Fanuc TP program (LS listing): JOB_VAR_ID_GRIP.LS

/PROG  JOB_VAR_ID_GRIP
/ATTR
OWNER		= MNEDITOR;
COMMENT		= "";
PROG_SIZE	= 104955;
CREATE		= DATE 19-07-31  TIME 17:01:20;
MODIFIED	= DATE 26-07-17  TIME 17:40:38;
FILE_NAME	= JOB_VARI;
VERSION		= 0;
LINE_COUNT = 3549;
MEMORY_SIZE	= 106079;
PROTECT		= READ_WRITE;
TCD:  STACK_SIZE	= 0,
      TASK_PRIORITY	= 50,
      TIME_SLICE	= 0,
      BUSY_LAMP_OFF	= 0,
      ABORT_REQUEST	= 0,
      PAUSE_REQUEST	= 0;
DEFAULT_GROUP	= 1,*,*,*,*;
CONTROL_CODE	= 00000000 00000000;
/APPL

AUTO_SINGULARITY_HEADER;
  ENABLE_SINGULARITY_AVOIDANCE   : TRUE;
/MN
   1:  !R[70] is the item number ;
   2:  !R[71] if using previous data ;
   3:  R[196]=AR[1]    ;
   4:  R[197]=AR[2]    ;
   5:  !------------------------- ;
   6:  !Item Select = 102610459 ;
   7:  SELECT R[70]=459,JMP LBL[459] ;
   8:  !Item Select = 102680512 ;
   9:         =512,JMP LBL[512] ;
  10:  !Item Select = 102730745 ;
  11:         =745,JMP LBL[745] ;
  12:  !Item Select = 102730746 ;
  13:         =746,JMP LBL[746] ;
  14:  !Item Select = 102730747 ;
  15:         =3074,JMP LBL[3074] ;
  16:  !Item Select = 102601361 ;
  17:         =1361,JMP LBL[1361] ;
  18:  !Item Select = 102601363 ;
  19:         =1363,JMP LBL[1363] ;
  20:  !Item Select = 102601364 ;
  21:         =1364,JMP LBL[1364] ;
  22:  !Item Select = 102601365 ;
  23:         =1365,JMP LBL[1365] ;
  24:  !Item Select = 102601366 ;
  25:         =1366,JMP LBL[1366] ;
  26:  !Item Select = 102601367 ;
  27:         =1367,JMP LBL[1367] ;
  28:  !Item Select = 102861623 ;
  29:         =1623,JMP LBL[1623] ;
  30:  !Item Select = 102681826 ;
  31:         =1826,JMP LBL[1826] ;
  32:  !Item Select = 102772047 ;
  33:         =2047,JMP LBL[2047] ;
  34:  !Item Select = 102772052 ;
  35:         =2052,JMP LBL[2052] ;
  36:  !Item Select = 103062126 ;
  37:         =2126,JMP LBL[2126] ;
  38:  !Item Select = 102592407 ;
  39:         =2407,JMP LBL[2407] ;
  40:  !Item Select = 102592408 ;
  41:         =2408,JMP LBL[2408] ;
  42:  !Item Select = 101463245 ;
  43:         =3245,JMP LBL[3245] ;
  44:  !Item Select = 102503284 ;
  45:         =3284,JMP LBL[3284] ;
  46:  !Item Select = 102703721 ;
  47:         =3721,JMP LBL[3721] ;
  48:  !Item Select = 102745613 ;
  49:         =5613,JMP LBL[5613] ;
  50:  !Item Select = 103205791 ;
  51:         =5791,JMP LBL[5791] ;
  52:  !Item Select = 100006970 ;
  53:         =6970,JMP LBL[6970] ;
  54:  !Item Select = 101487064 ;
  55:         =7064,JMP LBL[7064] ;
  56:  !Item Select = 101367132 ;
  57:         =7132,JMP LBL[7132] ;
  58:  !Item Select = 101477920 ;
  59:         =7920,JMP LBL[7920] ;
  60:  !Item Select = 101477937 ;
  61:         =7937,JMP LBL[7937] ;
  62:  !Item Select = 101444857 ;
  63:         =4857,JMP LBL[4857] ;
  64:  !Item Select = 103058815 ;
  65:         =8815,JMP LBL[8815] ;
  66:  !Item Select = 103209297 ;
  67:         =9297,JMP LBL[9297] ;
  68:  !Item Select = 102679394 ;
  69:         =9394,JMP LBL[9394] ;
  70:  !Item Select = 100009654 ;
  71:         =9654,JMP LBL[9654] ;
  72:  !Item Select = 1111199990 ;
  73:         =9990,JMP LBL[9990] ;
  74:  !No conditions are met, jump ;
  75:  !to the very end of the program ;
  76:         ELSE,JMP LBL[9999] ;
  77:   ;
  78:  LBL[459] ;
  79:  !--------------------------- ;
  80:  !Slip ;
  81:  !Item 102610459 , Rev D ;
  82:  !Last Modified: 2023-01-30 ;
  83:  !Modified by: Tsuu ;
  84:  !2.02 IN Height ;
  85:  !3.16 IN ID, 4.760 IN OD ;
  86:  !ID Jaw # 1025 ;
  87:  !--------------------------- ;
  88:  IF (R[70]=459) THEN ;
  89:   ;
  90:  !Define Parameters for INF/OTF ;
  91:  !R[105]=AR[1]=100, 2By3 Sheet ;
  92:  !R[105]=AR[1]=200, 3By4 Sheet ;
  93:  CALL JOB_VAR_SETUP(200) ;
  94:   ;
  95:  !--------------------------- ;
  96:  !Define Parameters for Job ;
  97:  !R[85] "INF_JAW_OFFSET"(Hgt) ;
  98:  R[85]=25    ;
  99:  !R[86] "INF_PICK_OFFSET" 50mm/sec ;
 100:  R[86]=13    ;
 101:  !R[87] "MAIN_LOAD_OFFSET" (PRELOA ;
 102:  R[87]=0    ;
 103:  !R[100] "GRIPPER_ID" 3 values ;
 104:  !If =100, ID Grippers Installed ;
 105:  !If =200, OD Grippers Installed ;
 106:  !If =300, OD 45 Degree Grippers ;
 107:  R[100]=100    ;
 108:  !--------------------------- ;
 109:   ;
 110:  !If using previous setup data ;
 111:  IF (R[71]=459) THEN ;
 112:   ;
 113:  !--------------------------- ;
 114:  !1st: Height of Raw piece ;
 115:  R[190]=53.848    ;
 116:  !2nd: Height of Finish piece ;
 117:  R[191]=51.308    ;
 118:  !3rd: Infeed Height Offset ;
 119:  R[192]=(-55)    ;
 120:  !4th: Outfeed Height Offset ;
 121:  R[193]=(-93)    ;
 122:  !--------------------------- ;
 123:   ;
 124:  CALL CREATE_REG(R[190],R[191],R[192],R[193]) ;
 125:   ;
 126:  ENDIF ;
 127:   ;
 128:  !If new loading or offloading pos ;
 129:  !SET R[104] "IMPORT_LOADPOS" ;
 130:  !SET R[104]=1000, Otherwise NO ;
 131:  R[104]=1000    ;
 132:  IF (R[104]=1000) THEN ;
 133:  !R[260]=43, Preload Pos1 ;
 134:  !R[270]=44, Preload PosFinal ;
 135:  !R[300]=53, Offload PosFinal ;
 136:  !PR[43] Pre-Loading Pos1 ;
 137:  CALL CREATE_PR(43,168.572,(-60.923),352.023,67.102,89.464,65.289) ;
 138:  !PR[44] Final Loading Position ;
 139:  CALL CREATE_PR(44,168.534,(-61.13),363.505,67.212,89.464,65.395) ;
 140:  !PR[53] pre-Unloading Position ;
 141:  CALL CREATE_PR(53,(-125.093),95.886,36.656,173.09,(-88.208),(-174.916)) ;
 142:  !PR[54] Final Unloading Position ;
 143:  CALL CREATE_PR(54,(-124.357),95.73,13.108,173.17,(-88.209),(-174.985)) ;
 144:  !PR[56] assitant Unloading preses ;
 145:  CALL CREATE_PR(56,(-133.84),95.467,273.686,(-177.134),(-88.249),175.184) ;
 146:  !PR[57] assitant Unloading preses ;
 147:  CALL CREATE_PR(57,(-135.964),108.085,344.284,(-177.144),(-88.245),175.194) ;
 148:  !PR[58] assitant Unloading preses ;
 149:  CALL CREATE_PR(58,296.854,360.959,378.47,(-91.75),(-.28),88.063) ;
 150:  ENDIF ;
 151:   ;
 152:  !---------------------------- ;
 153:  !SR[1] = "JOB_VAR_ID_GRIP" ;
 154:  !JOB_VAR_COMMON(R[103])'s value ;
 155:  !---------------------------- ;
 156:  !2By3 SR[1] INF, Max 18(Straight) ;
 157:  !R[103]=100 ;
 158:  !2By3 INF 45 Degree Diagonal Shif ;
 159:  !R[103]=110 ;
 160:  !---------------------------- ;
 161:  !3By4 SR[1] INF, Max 36(Straight) ;
 162:  !R[103]=150 ;
 163:  !3By4 INF 45 Degree Diagonal Shif ;
 164:  !R[103]=160 ;
 165:  !---------------------------- ;
 166:  !R[103] "JOB_PROFILE" Selection ;
 167:  R[103]=150    ;
 168:  CALL JOB_VAR_COMMON(R[103]) ;
 169:   ;
 170:  ENDIF ;
 171:   ;
 172:  JMP LBL[9999] ;
 173:   ;
 174:  !Job 102610459 Logic Ends ;
 175:  !--------------------------- ;
 176:   ;
 177:  LBL[512] ;
 178:  !--------------------------- ;
 179:  !Slip Carrier, Lower ;
 180:  !Item 102680512 , Rev A ;
 181:  !Last Modified: 2026-05-15 ;
 182:  !Modified by: Aaron ;
 183:  !3.74 IN Height ;
 184:  !3.150 IN ID, 4.500 IN OD, 6.0 Lb ;
 185:  !ID Jaw # 1010 ;
 186:  !--------------------------- ;
 187:  IF (R[70]=512) THEN ;
 188:   ;
 189:  !Define Parameters for INF/OTF ;
 190:  !R[105]=AR[1]=100, 2By3 Sheet ;
 191:  !R[105]=AR[1]=200, 3By4 Sheet ;
 192:  CALL JOB_VAR_SETUP(100) ;
 193:   ;
 194:  !--------------------------- ;
 195:  !Define Parameters for Job ;
 196:  R[1]=1    ;
 197:  R[2]=0    ;
 198:  R[4]=0    ;
 199:  R[67]=35    ;
 200:  !R[85] "INF_JAW_OFFSET"(Hgt) ;
 201:  R[85]=78.4    ;
 202:  !R[86] "INF_PICK_OFFSET" 50mm/sec ;
 203:  R[86]=10    ;
 204:  !R[87] "MAIN_LOAD_OFFSET" (PRELOA ;
 205:  R[87]=0    ;
 206:  !R[100] "GRIPPER_ID" 3 values ;
 207:  !If =100, ID Grippers Installed ;
 208:  !If =200, OD Grippers Installed ;
 209:  !If =300, OD 45 Degree Grippers ;
 210:  R[100]=100    ;
 211:  !--------------------------- ;
 212:   ;
 213:  !If using previous setup data ;
 214:  IF (R[71]=512) THEN ;
 215:   ;
 216:  !--------------------------- ;
 217:  !1st: Height of Raw piece ;
 218:  R[190]=101    ;
 219:  !2nd: Height of Finish piece ;
 220:  R[191]=95    ;
 221:  !3rd: Infeed Height Offset ;
 222:  R[192]=(-300)    ;
 223:  !4th: Outfeed Height Offset ;
 224:  R[193]=(-295)    ;
 225:  !--------------------------- ;
 226:   ;
 227:  CALL CREATE_REG(R[190],R[191],R[192],R[193]) ;
 228:   ;
 229:  ENDIF ;
 230:   ;
 231:  !If new loading or offloading pos ;
 232:  !SET R[104] "IMPORT_LOADPOS" ;
 233:  !SET R[104]=1000, Otherwise NO ;
 234:  R[104]=1000    ;
 235:  IF (R[104]=1000) THEN ;
 236:  !R[260]=43, Preload Pos1 ;
 237:  !R[270]=44, Preload PosFinal ;
 238:  !R[300]=53, Offload PosFinal ;
 239:  !PR[43] Pre-Loading Pos1 ;
 240:  CALL CREATE_PR(43,168.016,(-60.327),359.452,97.401,89.434,95.565) ;
 241:  !PR[44] Final Loading Position ;
 242:  CALL CREATE_PR(44,168.082,(-60.943),407.633,97.503,89.436,95.659) ;
 243:  !PR[53] pre-Unloading Position ;
 244:  CALL CREATE_PR(53,(-131.438),93.126,204.569,171.755,(-88.248),(-173.108)) ;
 245:  !PR[54] Final Unloading Position ;
 246:  CALL CREATE_PR(54,(-130.24),93.445,164.559,171.759,(-88.249),(-173.121)) ;
 247:  !PR[56] assitant Unloading preses ;
 248:  CALL CREATE_PR(56,(-133.84),95.467,273.686,(-177.134),(-88.249),175.184) ;
 249:  !PR[57] assitant Unloading preses ;
 250:  CALL CREATE_PR(57,(-135.964),108.085,344.284,(-177.144),(-88.245),175.194) ;
 251:  !PR[58] assitant Unloading preses ;
 252:  CALL CREATE_PR(58,296.854,360.959,378.47,(-91.75),(-.28),88.063) ;
 253:  ENDIF ;
 254:   ;
 255:  !---------------------------- ;
 256:  !SR[1] = "JOB_VAR_ID_GRIP" ;
 257:  !JOB_VAR_COMMON(R[103])'s value ;
 258:  !---------------------------- ;
 259:  !2By3 SR[1] INF, Max 18(Straight) ;
 260:  !R[103]=100 ;
 261:  !2By3 INF 45 Degree Diagonal Shif ;
 262:  !R[103]=110 ;
 263:  !---------------------------- ;
 264:  !3By4 SR[1] INF, Max 36(Straight) ;
 265:  !R[103]=150 ;
 266:  !3By4 INF 45 Degree Diagonal Shif ;
 267:  !R[103]=160 ;
 268:  !---------------------------- ;
 269:  !R[103] "JOB_PROFILE" Selection ;
 270:  R[103]=100    ;
 271:  CALL JOB_VAR_COMMON(R[103]) ;
 272:   ;
 273:  ENDIF ;
 274:   ;
 275:  JMP LBL[9999] ;
 276:   ;
 277:  !Job 102680512 Logic Ends ;
 278:  !--------------------------- ;
 279:   ;
 280:  LBL[745] ;
 281:  !--------------------------- ;
 282:  !Top Slip Support, Packer ;
 283:  !Item 102730745 , Rev A ;
 284:  !Last Modified: 2026-02-04 ;
 285:  !Modified by: Aaron ;
 286:  !4.705 IN Height ;
 287:  !3.4 IN ID, 4.18 IN OD, 18.5 Lbs ;
 288:  !ID Jaw # 1016 ;
 289:  !--------------------------- ;
 290:  IF (R[70]=745) THEN ;
 291:   ;
 292:  !Define Parameters for INF/OTF ;
 293:  !R[105]=AR[1]=100, 2By3 Sheet ;
 294:  !R[105]=AR[1]=200, 3By4 Sheet ;
 295:  CALL JOB_VAR_SETUP(100) ;
 296:   ;
 297:  !--------------------------- ;
 298:  !Define Parameters for Job ;
 299:  R[1]=1    ;
 300:  R[2]=1    ;
 301:  R[4]=0    ;
 302:  R[67]=45    ;
 303:  !R[85] "INF_JAW_OFFSET"(Hgt) ;
 304:  R[85]=20    ;
 305:  !R[86] "INF_PICK_OFFSET" 50mm/sec ;
 306:  R[86]=2    ;
 307:  !R[87] "MAIN_LOAD_OFFSET" (PRELOA ;
 308:  R[87]=0    ;
 309:  !R[100] "GRIPPER_ID" 3 values ;
 310:  !If =100, ID Grippers Installed ;
 311:  !If =200, OD Grippers Installed ;
 312:  !If =300, OD 45 Degree Grippers ;
 313:  R[100]=100    ;
 314:  !--------------------------- ;
 315:   ;
 316:  !If using previous setup data ;
 317:  IF (R[71]=745) THEN ;
 318:   ;
 319:  !--------------------------- ;
 320:  !1st: Height of Raw piece ;
 321:  R[190]=124.8    ;
 322:  !2nd: Height of Finish piece ;
 323:  R[191]=119.51    ;
 324:  !3rd: Infeed Height Offset ;
 325:  R[192]=(-298)    ;
 326:  !4th: Outfeed Height Offset ;
 327:  R[193]=(-250)    ;
 328:  !--------------------------- ;
 329:   ;
 330:  CALL CREATE_REG(R[190],R[191],R[192],R[193]) ;
 331:   ;
 332:  ENDIF ;
 333:   ;
 334:  !If new loading or offloading pos ;
 335:  !SET R[104] "IMPORT_LOADPOS" ;
 336:  !SET R[104]=1000, Otherwise NO ;
 337:  R[104]=1000    ;
 338:  IF (R[104]=1000) THEN ;
 339:  !R[260]=43, Preload Pos1 ;
 340:  !R[270]=44, Preload PosFinal ;
 341:  !R[300]=53, Offload PosFinal ;
 342:  !PR[43] Pre-Loading Pos1 ;
 343:  CALL CREATE_PR(43,163.322,(-60.984),274.82,151.418,88.347,149.991) ;
 344:  !PR[44] Final Loading Position ;
 345:  CALL CREATE_PR(44,164.891,(-62.061),335.467,151.455,88.338,150.017) ;
 346:  !PR[53] pre-Unloading Position ;
 347:  CALL CREATE_PR(53,(-130.787),93.777,177.177,170.605,(-88.218),(-171.87)) ;
 348:  !PR[54] Final Unloading Position ;
 349:  CALL CREATE_PR(54,(-127.959),94.047,84.786,170.695,(-88.22),(-171.955)) ;
 350:  !PR[56] assitant Unloading preses ;
 351:  CALL CREATE_PR(56,(-133.84),95.467,273.686,(-177.134),(-88.249),175.184) ;
 352:  !PR[57] assitant Unloading preses ;
 353:  CALL CREATE_PR(57,(-135.964),108.085,344.284,(-177.144),(-88.245),175.194) ;
 354:  !PR[58] assitant Unloading preses ;
 355:  CALL CREATE_PR(58,296.854,360.959,378.47,(-91.75),(-.28),88.063) ;
 356:  ENDIF ;
 357:   ;
 358:  !---------------------------- ;
 359:  !SR[1] = "JOB_VAR_ID_GRIP" ;
 360:  !JOB_VAR_COMMON(R[103])'s value ;
 361:  !---------------------------- ;
 362:  !2By3 SR[1] INF, Max 18(Straight) ;
 363:  !R[103]=100 ;
 364:  !2By3 INF 45 Degree Diagonal Shif ;
 365:  !R[103]=110 ;
 366:  !---------------------------- ;
 367:  !3By4 SR[1] INF, Max 36(Straight) ;
 368:  !R[103]=150 ;
 369:  !3By4 INF 45 Degree Diagonal Shif ;
 370:  !R[103]=160 ;
 371:  !---------------------------- ;
 372:  !R[103] "JOB_PROFILE" Selection ;
 373:  R[103]=100    ;
 374:  CALL JOB_VAR_COMMON(R[103]) ;
 375:   ;
 376:  ENDIF ;
 377:   ;
 378:  JMP LBL[9999] ;
 379:   ;
 380:  !Job 102730745 Logic Ends ;
 381:  !--------------------------- ;
 382:   ;
 383:  LBL[746] ;
 384:  !--------------------------- ;
 385:  !Wedge, Top ;
 386:  !Item 102730746 , Rev A ;
 387:  !Last Modified: 2026-05-04 ;
 388:  !Modified by: Aaron ;
 389:  !1.88 IN Height ;
 390:  !3.4 IN ID, 4.32 IN OD, 6.0 Lbs W ;
 391:  !ID Jaw # 1010 ;
 392:  !--------------------------- ;
 393:  IF (R[70]=746) THEN ;
 394:   ;
 395:  !Define Parameters for INF/OTF ;
 396:  !R[105]=AR[1]=100, 2By3 Sheet ;
 397:  !R[105]=AR[1]=200, 3By4 Sheet ;
 398:  CALL JOB_VAR_SETUP(100) ;
 399:   ;
 400:  !--------------------------- ;
 401:  !Define Parameters for Job ;
 402:  R[1]=1    ;
 403:  R[2]=1    ;
 404:  R[4]=0    ;
 405:  R[67]=10    ;
 406:  !R[85] "INF_JAW_OFFSET"(Hgt) ;
 407:  R[85]=94.4    ;
 408:  !R[86] "INF_PICK_OFFSET" 50mm/sec ;
 409:  R[86]=30    ;
 410:  !R[87] "MAIN_LOAD_OFFSET" (PRELOA ;
 411:  R[87]=0    ;
 412:  !R[100] "GRIPPER_ID" 3 values ;
 413:  !If =100, ID Grippers Installed ;
 414:  !If =200, OD Grippers Installed ;
 415:  !If =300, OD 45 Degree Grippers ;
 416:  R[100]=100    ;
 417:  !--------------------------- ;
 418:   ;
 419:  !If using previous setup data ;
 420:  IF (R[71]=746) THEN ;
 421:   ;
 422:  !--------------------------- ;
 423:  !1st: Height of Raw piece ;
 424:  R[190]=53.5    ;
 425:  !2nd: Height of Finish piece ;
 426:  R[191]=47.75    ;
 427:  !3rd: Infeed Height Offset ;
 428:  R[192]=(-300)    ;
 429:  !4th: Outfeed Height Offset ;
 430:  R[193]=(-295)    ;
 431:  !--------------------------- ;
 432:   ;
 433:  CALL CREATE_REG(R[190],R[191],R[192],R[193]) ;
 434:   ;
 435:  ENDIF ;
 436:   ;
 437:  !If new loading or offloading pos ;
 438:  !SET R[104] "IMPORT_LOADPOS" ;
 439:  !SET R[104]=1000, Otherwise NO ;
 440:  R[104]=1000    ;
 441:  IF (R[104]=1000) THEN ;
 442:  !R[260]=43, Preload Pos1 ;
 443:  !R[270]=44, Preload PosFinal ;
 444:  !R[300]=53, Offload PosFinal ;
 445:  !PR[43] Pre-Loading Pos1 ;
 446:  CALL CREATE_PR(43,168.016,(-60.327),359.452,97.401,89.434,95.565) ;
 447:  !PR[44] Final Loading Position ;
 448:  CALL CREATE_PR(44,168.082,(-60.943),407.633,97.503,89.436,95.659) ;
 449:  !PR[53] pre-Unloading Position ;
 450:  CALL CREATE_PR(53,(-131.438),93.126,204.569,171.755,(-88.248),(-173.108)) ;
 451:  !PR[54] Final Unloading Position ;
 452:  CALL CREATE_PR(54,(-130.24),93.445,164.559,171.759,(-88.249),(-173.121)) ;
 453:  !PR[56] assitant Unloading preses ;
 454:  CALL CREATE_PR(56,(-133.84),95.467,273.686,(-177.134),(-88.249),175.184) ;
 455:  !PR[57] assitant Unloading preses ;
 456:  CALL CREATE_PR(57,(-135.964),108.085,344.284,(-177.144),(-88.245),175.194) ;
 457:  !PR[58] assitant Unloading preses ;
 458:  CALL CREATE_PR(58,296.854,360.959,378.47,(-91.75),(-.28),88.063) ;
 459:  ENDIF ;
 460:   ;
 461:  !---------------------------- ;
 462:  !SR[1] = "JOB_VAR_ID_GRIP" ;
 463:  !JOB_VAR_COMMON(R[103])'s value ;
 464:  !---------------------------- ;
 465:  !2By3 SR[1] INF, Max 18(Straight) ;
 466:  !R[103]=100 ;
 467:  !2By3 INF 45 Degree Diagonal Shif ;
 468:  !R[103]=110 ;
 469:  !---------------------------- ;
 470:  !3By4 SR[1] INF, Max 36(Straight) ;
 471:  !R[103]=150 ;
 472:  !3By4 INF 45 Degree Diagonal Shif ;
 473:  !R[103]=160 ;
 474:  !---------------------------- ;
 475:  !R[103] "JOB_PROFILE" Selection ;
 476:  R[103]=100    ;
 477:  CALL JOB_VAR_COMMON(R[103]) ;
 478:   ;
 479:  ENDIF ;
 480:   ;
 481:  JMP LBL[9999] ;
 482:   ;
 483:  !Job 102730746 Logic Ends ;
 484:  !--------------------------- ;
 485:   ;
 486:  LBL[3074] ;
 487:  !--------------------------- ;
 488:  !Wedge, Bottom ;
 489:  !Item 102730747 , Rev A ;
 490:  !Last Modified: 2026-02-04 ;
 491:  !Modified by: Aaron ;
 492:  !2.1 IN Height ;
 493:  !3.4 IN ID, 4.3 IN OD, 9.0 Lbs W ;
 494:  !ID Jaw # 1010 ;
 495:  !--------------------------- ;
 496:  IF (R[70]=3074) THEN ;
 497:   ;
 498:  !Define Parameters for INF/OTF ;
 499:  !R[105]=AR[1]=100, 2By3 Sheet ;
 500:  !R[105]=AR[1]=200, 3By4 Sheet ;
 501:  CALL JOB_VAR_SETUP(100) ;
 502:   ;
 503:  !--------------------------- ;
 504:  !Define Parameters for Job ;
 505:  R[1]=1    ;
 506:  R[2]=1    ;
 507:  R[4]=0    ;
 508:  R[67]=15    ;
 509:  !R[85] "INF_JAW_OFFSET"(Hgt) ;
 510:  R[85]=20    ;
 511:  !R[86] "INF_PICK_OFFSET" 50mm/sec ;
 512:  R[86]=2    ;
 513:  !R[87] "MAIN_LOAD_OFFSET" (PRELOA ;
 514:  R[87]=0    ;
 515:  !R[100] "GRIPPER_ID" 3 values ;
 516:  !If =100, ID Grippers Installed ;
 517:  !If =200, OD Grippers Installed ;
 518:  !If =300, OD 45 Degree Grippers ;
 519:  R[100]=100    ;
 520:  !--------------------------- ;
 521:   ;
 522:  !If using previous setup data ;
 523:  IF (R[71]=3074) THEN ;
 524:   ;
 525:  !--------------------------- ;
 526:  !1st: Height of Raw piece ;
 527:  R[190]=59.69    ;
 528:  !2nd: Height of Finish piece ;
 529:  R[191]=53.34    ;
 530:  !3rd: Infeed Height Offset ;
 531:  R[192]=(-302)    ;
 532:  !4th: Outfeed Height Offset ;
 533:  R[193]=(-300)    ;
 534:  !--------------------------- ;
 535:   ;
 536:  CALL CREATE_REG(R[190],R[191],R[192],R[193]) ;
 537:   ;
 538:  ENDIF ;
 539:   ;
 540:  !If new loading or offloading pos ;
 541:  !SET R[104] "IMPORT_LOADPOS" ;
 542:  !SET R[104]=1000, Otherwise NO ;
 543:  R[104]=1000    ;
 544:  IF (R[104]=1000) THEN ;
 545:  !R[260]=43, Preload Pos1 ;
 546:  !R[270]=44, Preload PosFinal ;
 547:  !R[300]=53, Offload PosFinal ;
 548:  !PR[43] Pre-Loading Pos1 ;
 549:  CALL CREATE_PR(43,167.792,(-61.313),353.354,163.86,88.778,162.048) ;
 550:  !PR[44] Final Loading Position ;
 551:  CALL CREATE_PR(44,168.811,(-61.793),402.049,163.817,88.773,161.996) ;
 552:  !PR[53] pre-Unloading Position ;
 553:  CALL CREATE_PR(53,(-130.717),93.822,170.319,164.728,(-88.371),(-166.19)) ;
 554:  !PR[54] Final Unloading Position ;
 555:  CALL CREATE_PR(54,(-129.948),94.139,141.795,164.705,(-88.372),(-166.174)) ;
 556:  !PR[56] assitant Unloading preses ;
 557:  CALL CREATE_PR(56,(-133.84),95.467,273.686,(-177.134),(-88.249),175.184) ;
 558:  !PR[57] assitant Unloading preses ;
 559:  CALL CREATE_PR(57,(-135.964),108.085,344.284,(-177.144),(-88.245),175.194) ;
 560:  !PR[58] assitant Unloading preses ;
 561:  CALL CREATE_PR(58,296.854,360.959,378.47,(-91.75),(-.28),88.063) ;
 562:  ENDIF ;
 563:   ;
 564:  !---------------------------- ;
 565:  !SR[1] = "JOB_VAR_ID_GRIP" ;
 566:  !JOB_VAR_COMMON(R[103])'s value ;
 567:  !---------------------------- ;
 568:  !2By3 SR[1] INF, Max 18(Straight) ;
 569:  !R[103]=100 ;
 570:  !2By3 INF 45 Degree Diagonal Shif ;
 571:  !R[103]=110 ;
 572:  !---------------------------- ;
 573:  !3By4 SR[1] INF, Max 36(Straight) ;
 574:  !R[103]=150 ;
 575:  !3By4 INF 45 Degree Diagonal Shif ;
 576:  !R[103]=160 ;
 577:  !---------------------------- ;
 578:  !R[103] "JOB_PROFILE" Selection ;
 579:  R[103]=100    ;
 580:  CALL JOB_VAR_COMMON(R[103]) ;
 581:   ;
 582:  ENDIF ;
 583:   ;
 584:  JMP LBL[9999] ;
 585:   ;
 586:  !Job 102730747 Logic Ends ;
 587:  !--------------------------- ;
 588:   ;
 589:  LBL[1361] ;
 590:  !--------------------------- ;
 591:  !Ring,Spacer ;
 592:  !Item 102601361 , Rev A ;
 593:  !Last Modified: 2022-1-25 ;
 594:  !Modified by: Li ;
 595:  !0.5 IN Height ;
 596:  !2.4 IN ID, 3.68 IN OD ;
 597:  !ID Jaw # 1031 ;
 598:  !--------------------------- ;
 599:  IF (R[70]=1361) THEN ;
 600:   ;
 601:  !Define Parameters for INF/OTF ;
 602:  !R[105]=AR[1]=100, 2By3 Sheet ;
 603:  !R[105]=AR[1]=200, 3By4 Sheet ;
 604:  CALL JOB_VAR_SETUP(200) ;
 605:   ;
 606:  !--------------------------- ;
 607:  !Define Parameters for Job ;
 608:  !R[85] "INF_JAW_OFFSET"(Hgt) ;
 609:  R[85]=5    ;
 610:  !R[86] "INF_PICK_OFFSET" 50mm/sec ;
 611:  R[86]=1    ;
 612:  !R[87] "MAIN_LOAD_OFFSET" (PRELOA ;
 613:  R[87]=0    ;
 614:  !R[100] "GRIPPER_ID" 3 values ;
 615:  !If =100, ID Grippers Installed ;
 616:  !If =200, OD Grippers Installed ;
 617:  !If =300, OD 45 Degree Grippers ;
 618:  R[100]=100    ;
 619:  !--------------------------- ;
 620:   ;
 621:  !If using previous setup data ;
 622:  IF (R[71]=1361) THEN ;
 623:   ;
 624:  !--------------------------- ;
 625:  !1st: Height of Raw piece ;
 626:  R[190]=15.62    ;
 627:  !2nd: Height of Finish piece ;
 628:  R[191]=12.7    ;
 629:  !3rd: Infeed Height Offset ;
 630:  R[192]=(-15)    ;
 631:  !4th: Outfeed Height Offset ;
 632:  R[193]=(-60)    ;
 633:  !--------------------------- ;
 634:   ;
 635:  CALL CREATE_REG(R[190],R[191],R[192],R[193]) ;
 636:   ;
 637:  ENDIF ;
 638:   ;
 639:  !If new loading or offloading pos ;
 640:  !SET R[104] "IMPORT_LOADPOS" ;
 641:  !SET R[104]=1000, Otherwise NO ;
 642:  R[104]=1000    ;
 643:  IF (R[104]=1000) THEN ;
 644:  !R[260]=43, Preload Pos1 ;
 645:  !R[270]=44, Preload PosFinal ;
 646:  !R[300]=53, Offload PosFinal ;
 647:  !PR[43] Pre-Loading Pos1 ;
 648:  CALL CREATE_PR(43,168.672,(-60.32),286.786,19.084,88.42,17.227) ;
 649:  !PR[44] Final Loading Position ;
 650:  CALL CREATE_PR(44,168.515,(-60.14),296.211,19.111,88.421,17.247) ;
 651:  !PR[53] pre-Unloading Position ;
 652:  CALL CREATE_PR(53,(-131.629),93.837,242.229,172.716,(-88.209),(-174.573)) ;
 653:  !PR[54] Final Unloading Position ;
 654:  CALL CREATE_PR(54,(-131.414),93.939,234.768,172.696,(-88.211),(-174.558)) ;
 655:  !PR[56] assitant Unloading preses ;
 656:  CALL CREATE_PR(56,(-133.84),95.467,273.686,(-177.134),(-88.249),175.184) ;
 657:  !PR[57] assitant Unloading preses ;
 658:  CALL CREATE_PR(57,(-135.964),108.085,344.284,(-177.144),(-88.245),175.194) ;
 659:  !PR[58] assitant Unloading preses ;
 660:  CALL CREATE_PR(58,296.854,360.959,378.47,(-91.75),(-.28),88.063) ;
 661:  ENDIF ;
 662:   ;
 663:  !---------------------------- ;
 664:  !SR[1] = "JOB_VAR_ID_GRIP" ;
 665:  !JOB_VAR_COMMON(R[103])'s value ;
 666:  !---------------------------- ;
 667:  !2By3 SR[1] INF, Max 18(Straight) ;
 668:  !R[103]=100 ;
 669:  !2By3 INF 45 Degree Diagonal Shif ;
 670:  !R[103]=110 ;
 671:  !---------------------------- ;
 672:  !3By4 SR[1] INF, Max 36(Straight) ;
 673:  !R[103]=150 ;
 674:  !3By4 INF 45 Degree Diagonal Shif ;
 675:  !R[103]=160 ;
 676:  !---------------------------- ;
 677:  !R[103] "JOB_PROFILE" Selection ;
 678:  R[103]=150    ;
 679:  CALL JOB_VAR_COMMON(R[103]) ;
 680:   ;
 681:  ENDIF ;
 682:   ;
 683:  JMP LBL[9999] ;
 684:   ;
 685:  !Job 102601361 Logic Ends ;
 686:  !--------------------------- ;
 687:   ;
 688:  LBL[1363] ;
 689:  !--------------------------- ;
 690:  !Mandrel ;
 691:  !Item 102601363 , Rev xxx ;
 692:  !Last Modified: 2021-02-23 ;
 693:  !Modified by: Tsuu ;
 694:  !13.30 IN Height ;
 695:  !1.5 IN ID, 3.22 IN OD ;
 696:  !ID Jaw # Mandrel ;
 697:  !--------------------------- ;
 698:  IF (R[70]=1363) THEN ;
 699:   ;
 700:  !Define Parameters for INF/OTF ;
 701:  !R[105]=AR[1]=100, 2By3 Sheet ;
 702:  !R[105]=AR[1]=200, 3By4 Sheet ;
 703:  CALL JOB_VAR_SETUP(500) ;
 704:   ;
 705:  !--------------------------- ;
 706:  !Define Parameters for Job ;
 707:  !R[85] "INF_JAW_OFFSET"(Hgt) ;
 708:  R[85]=87.6    ;
 709:  !R[86] "INF_PICK_OFFSET" 50mm/sec ;
 710:  R[86]=20    ;
 711:  !R[87] "MAIN_LOAD_OFFSET" (PRELOA ;
 712:  R[87]=0    ;
 713:  !R[100] "GRIPPER_ID" 3 values ;
 714:  !If =100, ID Grippers Installed ;
 715:  !If =200, OD Grippers Installed ;
 716:  !If =300, OD 45 Degree Grippers ;
 717:  R[100]=100    ;
 718:  !--------------------------- ;
 719:   ;
 720:  !If using previous setup data ;
 721:  IF (R[71]=1363) THEN ;
 722:   ;
 723:  !--------------------------- ;
 724:  !1st: Height of Raw piece ;
 725:  R[190]=340    ;
 726:  !2nd: Height of Finish piece ;
 727:  R[191]=337.82    ;
 728:  !3rd: Infeed Height Offset ;
 729:  R[192]=(-65)    ;
 730:  !4th: Outfeed Height Offset ;
 731:  R[193]=(-176)    ;
 732:  !--------------------------- ;
 733:   ;
 734:  CALL CREATE_REG(R[190],R[191],R[192],R[193]) ;
 735:   ;
 736:  ENDIF ;
 737:   ;
 738:  !If new loading or offloading pos ;
 739:  !SET R[104] "IMPORT_LOADPOS" ;
 740:  !SET R[104]=1000, Otherwise NO ;
 741:  R[104]=1000    ;
 742:  IF (R[104]=1000) THEN ;
 743:  !R[260]=43, Preload Pos1 ;
 744:  !R[270]=44, Preload PosFinal ;
 745:  !R[300]=53, Offload PosFinal ;
 746:  !PR[43] Pre-Loading Pos1 ;
 747:  CALL CREATE_PR(43,167.168,(-70.982),(-9.637),153.289,88.751,151.207) ;
 748:  !PR[44] Final Loading Position ;
 749:  CALL CREATE_PR(44,170.064,(-70.749),137.992,157.287,88.784,155.172) ;
 750:  !PR[53] pre-Unloading Position ;
 751:  CALL CREATE_PR(53,(-132.181),108.408,216.873,173.351,(-88.246),(-175.317)) ;
 752:  !PR[54] Final Unloading Position ;
 753:  CALL CREATE_PR(54,(-127.477),109.006,61.614,173.251,(-88.248),(-175.226)) ;
 754:  !PR[56] assitant Unloading preses ;
 755:  CALL CREATE_PR(56,(-132.935),108.031,243.66,(-177.212),(-88.249),175.253) ;
 756:  !PR[57] assitant Unloading preses ;
 757:  CALL CREATE_PR(57,(-132.92),107.912,243.673,(-91.749),(-.28),88.057) ;
 758:  !PR[58] assitant Unloading preses ;
 759:  CALL CREATE_PR(58,296.854,360.959,378.47,(-91.75),(-.28),88.063) ;
 760:  ENDIF ;
 761:   ;
 762:  !---------------------------- ;
 763:  !SR[1] = "JOB_VAR_ID_GRIP" ;
 764:  !JOB_VAR_COMMON(R[103])'s value ;
 765:  !---------------------------- ;
 766:  !2By3 SR[1] INF, Max 18(Straight) ;
 767:  !R[103]=100 ;
 768:  !2By3 INF 45 Degree Diagonal Shif ;
 769:  !R[103]=110 ;
 770:  !---------------------------- ;
 771:  !3By4 SR[1] INF, Max 36(Straight) ;
 772:  !R[103]=150 ;
 773:  !3By4 INF 45 Degree Diagonal Shif ;
 774:  !R[103]=160 ;
 775:  !---------------------------- ;
 776:  !R[103] "JOB_PROFILE" Selection ;
 777:  R[103]=160    ;
 778:  CALL JOB_VAR_COMMON(R[103]) ;
 779:   ;
 780:  ENDIF ;
 781:   ;
 782:  JMP LBL[9999] ;
 783:   ;
 784:  !Job 102601363 Logic Ends ;
 785:  !--------------------------- ;
 786:   ;
 787:  LBL[1364] ;
 788:  !--------------------------- ;
 789:  !Ring,Spacer ;
 790:  !Item 102601364 , Rev A ;
 791:  !Last Modified: 2021-10-19 ;
 792:  !Modified by: Tsuu ;
 793:  !0.5 IN Height ;
 794:  !2.4 IN ID, 3.68 IN OD ;
 795:  !ID Jaw # 1031 ;
 796:  !--------------------------- ;
 797:  IF (R[70]=1364) THEN ;
 798:   ;
 799:  !Define Parameters for INF/OTF ;
 800:  !R[105]=AR[1]=100, 2By3 Sheet ;
 801:  !R[105]=AR[1]=200, 3By4 Sheet ;
 802:  CALL JOB_VAR_SETUP(200) ;
 803:   ;
 804:  !--------------------------- ;
 805:  !Define Parameters for Job ;
 806:  !R[85] "INF_JAW_OFFSET"(Hgt) ;
 807:  R[85]=5    ;
 808:  !R[86] "INF_PICK_OFFSET" 50mm/sec ;
 809:  R[86]=1    ;
 810:  !R[87] "MAIN_LOAD_OFFSET" (PRELOA ;
 811:  R[87]=0    ;
 812:  !R[100] "GRIPPER_ID" 3 values ;
 813:  !If =100, ID Grippers Installed ;
 814:  !If =200, OD Grippers Installed ;
 815:  !If =300, OD 45 Degree Grippers ;
 816:  R[100]=100    ;
 817:  !--------------------------- ;
 818:   ;
 819:  !If using previous setup data ;
 820:  IF (R[71]=1364) THEN ;
 821:   ;
 822:  !--------------------------- ;
 823:  !1st: Height of Raw piece ;
 824:  R[190]=15.62    ;
 825:  !2nd: Height of Finish piece ;
 826:  R[191]=12.7    ;
 827:  !3rd: Infeed Height Offset ;
 828:  R[192]=(-15)    ;
 829:  !4th: Outfeed Height Offset ;
 830:  R[193]=(-60)    ;
 831:  !--------------------------- ;
 832:   ;
 833:  CALL CREATE_REG(R[190],R[191],R[192],R[193]) ;
 834:   ;
 835:  ENDIF ;
 836:   ;
 837:  !If new loading or offloading pos ;
 838:  !SET R[104] "IMPORT_LOADPOS" ;
 839:  !SET R[104]=1000, Otherwise NO ;
 840:  R[104]=1000    ;
 841:  IF (R[104]=1000) THEN ;
 842:  !R[260]=43, Preload Pos1 ;
 843:  !R[270]=44, Preload PosFinal ;
 844:  !R[300]=53, Offload PosFinal ;
 845:  !PR[43] Pre-Loading Pos1 ;
 846:  CALL CREATE_PR(43,168.672,(-60.32),286.786,19.084,88.42,17.227) ;
 847:  !PR[44] Final Loading Position ;
 848:  CALL CREATE_PR(44,168.515,(-60.14),296.211,19.111,88.421,17.247) ;
 849:  !PR[53] pre-Unloading Position ;
 850:  CALL CREATE_PR(53,(-131.629),93.837,242.229,172.716,(-88.209),(-174.573)) ;
 851:  !PR[54] Final Unloading Position ;
 852:  CALL CREATE_PR(54,(-131.414),93.939,234.768,172.696,(-88.211),(-174.558)) ;
 853:  !PR[56] assitant Unloading preses ;
 854:  CALL CREATE_PR(56,(-133.84),95.467,273.686,(-177.134),(-88.249),175.184) ;
 855:  !PR[57] assitant Unloading preses ;
 856:  CALL CREATE_PR(57,(-135.964),108.085,344.284,(-177.144),(-88.245),175.194) ;
 857:  !PR[58] assitant Unloading preses ;
 858:  CALL CREATE_PR(58,296.854,360.959,378.47,(-91.75),(-.28),88.063) ;
 859:  ENDIF ;
 860:   ;
 861:  !---------------------------- ;
 862:  !SR[1] = "JOB_VAR_ID_GRIP" ;
 863:  !JOB_VAR_COMMON(R[103])'s value ;
 864:  !---------------------------- ;
 865:  !2By3 SR[1] INF, Max 18(Straight) ;
 866:  !R[103]=100 ;
 867:  !2By3 INF 45 Degree Diagonal Shif ;
 868:  !R[103]=110 ;
 869:  !---------------------------- ;
 870:  !3By4 SR[1] INF, Max 36(Straight) ;
 871:  !R[103]=150 ;
 872:  !3By4 INF 45 Degree Diagonal Shif ;
 873:  !R[103]=160 ;
 874:  !---------------------------- ;
 875:  !R[103] "JOB_PROFILE" Selection ;
 876:  R[103]=150    ;
 877:  CALL JOB_VAR_COMMON(R[103]) ;
 878:   ;
 879:  ENDIF ;
 880:   ;
 881:  JMP LBL[9999] ;
 882:   ;
 883:  !Job 102601364 Logic Ends ;
 884:  !--------------------------- ;
 885:   ;
 886:  LBL[1365] ;
 887:  !--------------------------- ;
 888:  !SLIP, BUTTON ;
 889:  !Item 102601365 , Rev C ;
 890:  !Last Modified: 2023-10-10 ;
 891:  !Modified by: SH ;
 892:  !1.85 IN Height ;
 893:  !2.860 IN ID, 3.900 IN OD ;
 894:  !ID Jaw # 1025 ;
 895:  !--------------------------- ;
 896:  IF (R[70]=1365) THEN ;
 897:   ;
 898:  !Define Parameters for INF/OTF ;
 899:  !R[105]=AR[1]=100, 2By3 Sheet ;
 900:  !R[105]=AR[1]=200, 3By4 Sheet ;
 901:  CALL JOB_VAR_SETUP(200) ;
 902:   ;
 903:  !--------------------------- ;
 904:  !Define Parameters for Job ;
 905:  !R[85] "INF_JAW_OFFSET"(Hgt) ;
 906:  R[85]=25    ;
 907:  !R[86] "INF_PICK_OFFSET" 50mm/sec ;
 908:  R[86]=13    ;
 909:  !R[87] "MAIN_LOAD_OFFSET" (PRELOA ;
 910:  R[87]=0    ;
 911:  !R[100] "GRIPPER_ID" 3 values ;
 912:  !If =100, ID Grippers Installed ;
 913:  !If =200, OD Grippers Installed ;
 914:  !If =300, OD 45 Degree Grippers ;
 915:  R[100]=100    ;
 916:  !--------------------------- ;
 917:   ;
 918:  !If using previous setup data ;
 919:  IF (R[71]=1365) THEN ;
 920:   ;
 921:  !--------------------------- ;
 922:  !1st: Height of Raw piece ;
 923:  R[190]=52.07    ;
 924:  !2nd: Height of Finish piece ;
 925:  R[191]=46.99    ;
 926:  !3rd: Infeed Height Offset ;
 927:  R[192]=(-55)    ;
 928:  !4th: Outfeed Height Offset ;
 929:  R[193]=(-75)    ;
 930:  !--------------------------- ;
 931:   ;
 932:  CALL CREATE_REG(R[190],R[191],R[192],R[193]) ;
 933:   ;
 934:  ENDIF ;
 935:   ;
 936:  !If new loading or offloading pos ;
 937:  !SET R[104] "IMPORT_LOADPOS" ;
 938:  !SET R[104]=1000, Otherwise NO ;
 939:  R[104]=1000    ;
 940:  IF (R[104]=1000) THEN ;
 941:  !R[260]=43, Preload Pos1 ;
 942:  !R[270]=44, Preload PosFinal ;
 943:  !R[300]=53, Offload PosFinal ;
 944:  !PR[43] Pre-Loading Pos1 ;
 945:  CALL CREATE_PR(43,168.392,(-60.421),355.25,94.092,89.323,92.248) ;
 946:  !PR[44] Final Loading Position ;
 947:  CALL CREATE_PR(44,168.417,(-60.689),368.273,94.21,89.324,92.362) ;
 948:  !PR[53] pre-Unloading Position ;
 949:  CALL CREATE_PR(53,(-126.657),95.026,87.416,171.082,(-88.272),(-172.862)) ;
 950:  !PR[54] Final Unloading Position ;
 951:  CALL CREATE_PR(54,(-128.901),94.159,54.028,167.264,(-89.083),(-168.974)) ;
 952:  !PR[56] assitant Unloading preses ;
 953:  CALL CREATE_PR(56,(-133.84),95.467,273.686,(-177.134),(-88.249),175.184) ;
 954:  !PR[57] assitant Unloading preses ;
 955:  CALL CREATE_PR(57,(-135.964),108.085,344.284,(-177.144),(-88.245),175.194) ;
 956:  !PR[58] assitant Unloading preses ;
 957:  CALL CREATE_PR(58,296.854,360.959,378.47,(-91.75),(-.28),88.063) ;
 958:  ENDIF ;
 959:   ;
 960:  !---------------------------- ;
 961:  !SR[1] = "JOB_VAR_ID_GRIP" ;
 962:  !JOB_VAR_COMMON(R[103])'s value ;
 963:  !---------------------------- ;
 964:  !2By3 SR[1] INF, Max 18(Straight) ;
 965:  !R[103]=100 ;
 966:  !---------------------------- ;
 967:  !3By4 SR[1] INF, Max 36(Straight) ;
 968:  !R[103]=150 ;
 969:  !---------------------------- ;
 970:  !R[103] "JOB_PROFILE" Selection ;
 971:  R[103]=150    ;
 972:  CALL JOB_VAR_COMMON(R[103]) ;
 973:   ;
 974:  ENDIF ;
 975:   ;
 976:  JMP LBL[9999] ;
 977:   ;
 978:  !Job 102601365 Logic Ends ;
 979:  !--------------------------- ;
 980:   ;
 981:  LBL[1366] ;
 982:  !--------------------------- ;
 983:  !Wedge ;
 984:  !Item 102601366 , Rev B ;
 985:  !Last Modified: 2022-12-06 ;
 986:  !Modified by: Tsuu ;
 987:  !1.86 IN Height ;
 988:  !2.395 IN ID, 3.55 IN OD ;
 989:  !ID Jaw # 1031 ;
 990:  !--------------------------- ;
 991:  IF (R[70]=1366) THEN ;
 992:   ;
 993:  !Define Parameters for INF/OTF ;
 994:  !R[105]=AR[1]=100, 2By3 Sheet ;
 995:  !R[105]=AR[1]=200, 3By4 Sheet ;
 996:  CALL JOB_VAR_SETUP(200) ;
 997:   ;
 998:  !--------------------------- ;
 999:  !Define Parameters for Job ;
1000:  !R[85] "INF_JAW_OFFSET"(Hgt) ;
1001:  R[85]=10    ;
1002:  !R[86] "INF_PICK_OFFSET" 50mm/sec ;
1003:  R[86]=5    ;
1004:  !R[87] "MAIN_LOAD_OFFSET" (PRELOA ;
1005:  R[87]=0    ;
1006:  !R[100] "GRIPPER_ID" 3 values ;
1007:  !If =100, ID Grippers Installed ;
1008:  !If =200, OD Grippers Installed ;
1009:  !If =300, OD 45 Degree Grippers ;
1010:  R[100]=100    ;
1011:  !--------------------------- ;
1012:   ;
1013:  !If using previous setup data ;
1014:  IF (R[71]=1366) THEN ;
1015:   ;
1016:  !--------------------------- ;
1017:  !1st: Height of Raw piece ;
1018:  R[190]=49.5    ;
1019:  !2nd: Height of Finish piece ;
1020:  R[191]=47.24    ;
1021:  !3rd: Infeed Height Offset ;
1022:  R[192]=(-12)    ;
1023:  !4th: Outfeed Height Offset ;
1024:  !Changing 1st Level Offset to ;
1025:  R[193]=(-39)    ;
1026:   ;
1027:  !Changing 2nd Level Offset to ;
1028:  R[194]=(-41)    ;
1029:   ;
1030:  !Changing 3rd Level Offset to ;
1031:  R[195]=(-44)    ;
1032:   ;
1033:  CALL GN_OUTFEED_COMPENSATE(R[193],R[194],R[195]) ;
1034:  !--------------------------- ;
1035:   ;
1036:  CALL CREATE_REG(R[190],R[191],R[192],R[193]) ;
1037:   ;
1038:  ENDIF ;
1039:   ;
1040:  !If new loading or offloading pos ;
1041:  !SET R[104] "IMPORT_LOADPOS" ;
1042:  !SET R[104]=1000, Otherwise NO ;
1043:  R[104]=1000    ;
1044:  IF (R[104]=1000) THEN ;
1045:  !R[260]=43, Preload Pos1 ;
1046:  !R[270]=44, Preload PosFinal ;
1047:  !R[300]=53, Offload PosFinal ;
1048:  !PR[43] Pre-Loading Pos1 ;
1049:  CALL CREATE_PR(43,168.595,(-60.02),314.259,39.257,88.966,37.465) ;
1050:  !PR[44] Final Loading Position ;
1051:  CALL CREATE_PR(44,168.455,(-60.224),325.065,39.2,88.966,37.402) ;
1052:  !PR[53] pre-Unloading Position ;
1053:  CALL CREATE_PR(53,(-126.556),94.087,78.828,172.81,(-88.213),(-174.658)) ;
1054:  !PR[54] Final Unloading Position ;
1055:  CALL CREATE_PR(54,(-125.525),94.282,45.231,172.814,(-88.213),(-174.667)) ;
1056:  !PR[56] assitant Unloading preses ;
1057:  CALL CREATE_PR(56,(-133.84),95.467,273.686,(-177.134),(-88.249),175.184) ;
1058:  !PR[57] assitant Unloading preses ;
1059:  CALL CREATE_PR(57,(-135.964),108.085,344.284,(-177.144),(-88.245),175.194) ;
1060:  !PR[58] assitant Unloading preses ;
1061:  CALL CREATE_PR(58,296.854,360.959,378.47,(-91.75),(-.28),88.063) ;
1062:  ENDIF ;
1063:   ;
1064:  !---------------------------- ;
1065:  !SR[1] = "JOB_VAR_ID_GRIP" ;
1066:  !JOB_VAR_COMMON(R[103])'s value ;
1067:  !---------------------------- ;
1068:  !2By3 SR[1] INF, Max 18(Straight) ;
1069:  !R[103]=100 ;
1070:  !2By3 INF 45 Degree Diagonal Shif ;
1071:  !R[103]=110 ;
1072:  !---------------------------- ;
1073:  !3By4 SR[1] INF, Max 36(Straight) ;
1074:  !R[103]=150 ;
1075:  !3By4 INF 45 Degree Diagonal Shif ;
1076:  !R[103]=160 ;
1077:  !---------------------------- ;
1078:  !R[103] "JOB_PROFILE" Selection ;
1079:  R[103]=150    ;
1080:  CALL JOB_VAR_COMMON(R[103]) ;
1081:   ;
1082:  ENDIF ;
1083:   ;
1084:  JMP LBL[9999] ;
1085:   ;
1086:  !Job 102601366 Logic Ends ;
1087:  !--------------------------- ;
1088:   ;
1089:  LBL[1367] ;
1090:  !--------------------------- ;
1091:  !SLIP, BUTTON ;
1092:  !Item 102601367 , Rev D ;
1093:  !Last Modified: 2023-09-15 ;
1094:  !Modified by: Tsuu ;
1095:  !1.85 IN Height ;
1096:  !2.860 IN ID, 3.900 IN OD ;
1097:  !ID Jaw # 1025 ;
1098:  !--------------------------- ;
1099:  IF (R[70]=1367) THEN ;
1100:   ;
1101:  !Define Parameters for INF/OTF ;
1102:  !R[105]=AR[1]=100, 2By3 Sheet ;
1103:  !R[105]=AR[1]=200, 3By4 Sheet ;
1104:  CALL JOB_VAR_SETUP(200) ;
1105:   ;
1106:  !--------------------------- ;
1107:  !Define Parameters for Job ;
1108:  !R[85] "INF_JAW_OFFSET"(Hgt) ;
1109:  R[85]=25    ;
1110:  !R[86] "INF_PICK_OFFSET" 50mm/sec ;
1111:  R[86]=13    ;
1112:  !R[87] "MAIN_LOAD_OFFSET" (PRELOA ;
1113:  R[87]=0    ;
1114:  !R[100] "GRIPPER_ID" 3 values ;
1115:  !If =100, ID Grippers Installed ;
1116:  !If =200, OD Grippers Installed ;
1117:  !If =300, OD 45 Degree Grippers ;
1118:  R[100]=100    ;
1119:  !--------------------------- ;
1120:   ;
1121:  !If using previous setup data ;
1122:  IF (R[71]=1367) THEN ;
1123:   ;
1124:  !--------------------------- ;
1125:  !1st: Height of Raw piece ;
1126:  R[190]=52.07    ;
1127:  !2nd: Height of Finish piece ;
1128:  R[191]=46.99    ;
1129:  !3rd: Infeed Height Offset ;
1130:  R[192]=(-55)    ;
1131:  !4th: Outfeed Height Offset ;
1132:  R[193]=(-95)    ;
1133:  !--------------------------- ;
1134:   ;
1135:  CALL CREATE_REG(R[190],R[191],R[192],R[193]) ;
1136:   ;
1137:  ENDIF ;
1138:   ;
1139:  !If new loading or offloading pos ;
1140:  !SET R[104] "IMPORT_LOADPOS" ;
1141:  !SET R[104]=1000, Otherwise NO ;
1142:  R[104]=1000    ;
1143:  IF (R[104]=1000) THEN ;
1144:  !R[260]=43, Preload Pos1 ;
1145:  !R[270]=44, Preload PosFinal ;
1146:  !R[300]=53, Offload PosFinal ;
1147:  !PR[43] Pre-Loading Pos1 ;
1148:  CALL CREATE_PR(43,168.392,(-60.421),355.25,94.092,89.323,92.248) ;
1149:  !PR[44] Final Loading Position ;
1150:  CALL CREATE_PR(44,168.417,(-60.689),368.273,94.21,89.324,92.362) ;
1151:  !PR[53] pre-Unloading Position ;
1152:  CALL CREATE_PR(53,(-126.657),95.026,87.416,171.082,(-88.272),(-172.862)) ;
1153:  !PR[54] Final Unloading Position ;
1154:  CALL CREATE_PR(54,(-128.901),94.159,54.028,167.264,(-89.083),(-168.974)) ;
1155:  !PR[56] assitant Unloading preses ;
1156:  CALL CREATE_PR(56,(-133.84),95.467,273.686,(-177.134),(-88.249),175.184) ;
1157:  !PR[57] assitant Unloading preses ;
1158:  CALL CREATE_PR(57,(-135.964),108.085,344.284,(-177.144),(-88.245),175.194) ;
1159:  !PR[58] assitant Unloading preses ;
1160:  CALL CREATE_PR(58,296.854,360.959,378.47,(-91.75),(-.28),88.063) ;
1161:  ENDIF ;
1162:   ;
1163:  !---------------------------- ;
1164:  !SR[1] = "JOB_VAR_ID_GRIP" ;
1165:  !JOB_VAR_COMMON(R[103])'s value ;
1166:  !---------------------------- ;
1167:  !2By3 SR[1] INF, Max 18(Straight) ;
1168:  !R[103]=100 ;
1169:  !---------------------------- ;
1170:  !3By4 SR[1] INF, Max 36(Straight) ;
1171:  !R[103]=150 ;
1172:  !---------------------------- ;
1173:  !R[103] "JOB_PROFILE" Selection ;
1174:  R[103]=150    ;
1175:  CALL JOB_VAR_COMMON(R[103]) ;
1176:   ;
1177:  ENDIF ;
1178:   ;
1179:  JMP LBL[9999] ;
1180:   ;
1181:  !Job 102601367 Logic Ends ;
1182:  !--------------------------- ;
1183:   ;
1184:  LBL[1623] ;
1185:  !--------------------------- ;
1186:  !Slip ;
1187:  !Item 102861623 , Rev C ;
1188:  !Last Modified: 2023-01-31 ;
1189:  !Modified by: Tsuu ;
1190:  !1.89 IN Height ;
1191:  !2.550 IN ID, 3.950 IN OD ;
1192:  !ID Jaw # 1025 ;
1193:  !--------------------------- ;
1194:  IF (R[70]=1623) THEN ;
1195:   ;
1196:  !Define Parameters for INF/OTF ;
1197:  !R[105]=AR[1]=100, 2By3 Sheet ;
1198:  !R[105]=AR[1]=200, 3By4 Sheet ;
1199:  CALL JOB_VAR_SETUP(200) ;
1200:   ;
1201:  !--------------------------- ;
1202:  !Define Parameters for Job ;
1203:  !R[85] "INF_JAW_OFFSET"(Hgt) ;
1204:  R[85]=25    ;
1205:  !R[86] "INF_PICK_OFFSET" 50mm/sec ;
1206:  R[86]=13    ;
1207:  !R[87] "MAIN_LOAD_OFFSET" (PRELOA ;
1208:  R[87]=0    ;
1209:  !R[100] "GRIPPER_ID" 3 values ;
1210:  !If =100, ID Grippers Installed ;
1211:  !If =200, OD Grippers Installed ;
1212:  !If =300, OD 45 Degree Grippers ;
1213:  R[100]=100    ;
1214:  !--------------------------- ;
1215:   ;
1216:  !If using previous setup data ;
1217:  IF (R[71]=1623) THEN ;
1218:   ;
1219:  !--------------------------- ;
1220:  !1st: Height of Raw piece ;
1221:  R[190]=50.84    ;
1222:  !2nd: Height of Finish piece ;
1223:  R[191]=48.006    ;
1224:  !3rd: Infeed Height Offset ;
1225:  R[192]=(-55)    ;
1226:  !4th: Outfeed Height Offset ;
1227:  R[193]=(-80)    ;
1228:  !--------------------------- ;
1229:   ;
1230:  CALL CREATE_REG(R[190],R[191],R[192],R[193]) ;
1231:   ;
1232:  ENDIF ;
1233:   ;
1234:  !If new loading or offloading pos ;
1235:  !SET R[104] "IMPORT_LOADPOS" ;
1236:  !SET R[104]=1000, Otherwise NO ;
1237:  R[104]=1000    ;
1238:  IF (R[104]=1000) THEN ;
1239:  !R[260]=43, Preload Pos1 ;
1240:  !R[270]=44, Preload PosFinal ;
1241:  !R[300]=53, Offload PosFinal ;
1242:  !PR[43] Pre-Loading Pos1 ;
1243:  CALL CREATE_PR(43,168.573,(-60.592),357.506,67.647,89.471,65.85) ;
1244:  !PR[44] Final Loading Position ;
1245:  CALL CREATE_PR(44,168.559,(-61.792),366.433,67.955,89.471,66.152) ;
1246:  !PR[53] pre-Unloading Position ;
1247:  CALL CREATE_PR(53,(-125.816),95.978,70.546,171.289,(-88.225),(-173.093)) ;
1248:  !PR[54] Final Unloading Position ;
1249:  CALL CREATE_PR(54,(-124.965),95.019,43.083,171.848,(-88.22),(-173.644)) ;
1250:  !PR[56] assitant Unloading preses ;
1251:  CALL CREATE_PR(56,(-133.84),95.467,273.686,(-177.134),(-88.249),175.184) ;
1252:  !PR[57] assitant Unloading preses ;
1253:  CALL CREATE_PR(57,(-135.964),108.085,344.284,(-177.144),(-88.245),175.194) ;
1254:  !PR[58] assitant Unloading preses ;
1255:  CALL CREATE_PR(58,296.854,360.959,378.47,(-91.75),(-.28),88.063) ;
1256:  ENDIF ;
1257:   ;
1258:  !---------------------------- ;
1259:  !SR[1] = "JOB_VAR_ID_GRIP" ;
1260:  !JOB_VAR_COMMON(R[103])'s value ;
1261:  !---------------------------- ;
1262:  !2By3 SR[1] INF, Max 18(Straight) ;
1263:  !R[103]=100 ;
1264:  !2By3 INF 45 Degree Diagonal Shif ;
1265:  !R[103]=110 ;
1266:  !---------------------------- ;
1267:  !3By4 SR[1] INF, Max 36(Straight) ;
1268:  !R[103]=150 ;
1269:  !3By4 INF 45 Degree Diagonal Shif ;
1270:  !R[103]=160 ;
1271:  !---------------------------- ;
1272:  !R[103] "JOB_PROFILE" Selection ;
1273:  R[103]=150    ;
1274:  CALL JOB_VAR_COMMON(R[103]) ;
1275:   ;
1276:  ENDIF ;
1277:   ;
1278:  JMP LBL[9999] ;
1279:   ;
1280:  !Job 102861623 Logic Ends ;
1281:  !--------------------------- ;
1282:   ;
1283:  !--------------------------- ;
1284:  LBL[1826] ;
1285:  !--------------------------- ;
1286:  !Ring,Spacer ;
1287:  !Item 102681826 , Rev A ;
1288:  !Last Modified: 2023-08-31 ;
1289:  !Modified by: Tsuu ;
1290:  !0.5 IN Height ;
1291:  !2.400 IN ID, 3.68 IN OD ;
1292:  !ID Jaw # 1032 ;
1293:  !--------------------------- ;
1294:  IF (R[70]=1826) THEN ;
1295:   ;
1296:  !Define Parameters for INF/OTF ;
1297:  !R[105]=AR[1]=100, 2By3 Sheet ;
1298:  !R[105]=AR[1]=200, 3By4 Sheet ;
1299:  CALL JOB_VAR_SETUP(200) ;
1300:   ;
1301:  !--------------------------- ;
1302:  !Define Parameters for Job ;
1303:  !R[85] "INF_JAW_OFFSET"(Hgt) ;
1304:  R[85]=5    ;
1305:  !R[86] "INF_PICK_OFFSET" 50mm/sec ;
1306:  R[86]=1    ;
1307:  !R[87] "MAIN_LOAD_OFFSET" (PRELOA ;
1308:  R[87]=0    ;
1309:  !R[100] "GRIPPER_ID" 3 values ;
1310:  !If =100, ID Grippers Installed ;
1311:  !If =200, OD Grippers Installed ;
1312:  !If =300, OD 45 Degree Grippers ;
1313:  R[100]=100    ;
1314:  !--------------------------- ;
1315:   ;
1316:  !If using previous setup data ;
1317:  IF (R[71]=1826) THEN ;
1318:   ;
1319:  !--------------------------- ;
1320:  !1st: Height of Raw piece ;
1321:  R[190]=15.62    ;
1322:  !2nd: Height of Finish piece ;
1323:  R[191]=12.7    ;
1324:  !3rd: Infeed Height Offset ;
1325:  R[192]=(-16)    ;
1326:  !4th: Outfeed Height Offset ;
1327:  R[193]=(-57)    ;
1328:  !--------------------------- ;
1329:   ;
1330:  CALL CREATE_REG(R[190],R[191],R[192],R[193]) ;
1331:   ;
1332:  ENDIF ;
1333:   ;
1334:  !If new loading or offloading pos ;
1335:  !SET R[104] "IMPORT_LOADPOS" ;
1336:  !SET R[104]=1000, Otherwise NO ;
1337:  R[104]=1000    ;
1338:  IF (R[104]=1000) THEN ;
1339:  !R[260]=43, Preload Pos1 ;
1340:  !R[270]=44, Preload PosFinal ;
1341:  !R[300]=53, Offload PosFinal ;
1342:  !PR[43] Pre-Loading Pos1 ;
1343:  CALL CREATE_PR(43,169.417,(-60.156),283.549,19.611,88.443,17.772) ;
1344:  !PR[44] Final Loading Position ;
1345:  CALL CREATE_PR(44,169.095,(-60.369),296.57,19.628,88.445,17.784) ;
1346:  !PR[53] pre-Unloading Position ;
1347:  CALL CREATE_PR(53,(-131.629),93.837,242.229,172.716,(-88.209),(-174.573)) ;
1348:  !PR[54] Final Unloading Position ;
1349:  CALL CREATE_PR(54,(-131.424),93.782,234.425,172.817,(-88.215),(-174.673)) ;
1350:  !PR[56] assitant Unloading preses ;
1351:  CALL CREATE_PR(56,(-133.84),95.467,273.686,(-177.134),(-88.249),175.184) ;
1352:  !PR[57] assitant Unloading preses ;
1353:  CALL CREATE_PR(57,(-135.964),108.085,344.284,(-177.144),(-88.245),175.194) ;
1354:  !PR[58] assitant Unloading preses ;
1355:  CALL CREATE_PR(58,296.854,360.959,378.47,(-91.75),(-.28),88.063) ;
1356:  ENDIF ;
1357:   ;
1358:  !---------------------------- ;
1359:  !SR[1] = "JOB_VAR_ID_GRIP" ;
1360:  !JOB_VAR_COMMON(R[103])'s value ;
1361:  !---------------------------- ;
1362:  !2By3 SR[1] INF, Max 18(Straight) ;
1363:  !R[103]=100 ;
1364:  !2By3 INF 45 Degree Diagonal Shif ;
1365:  !R[103]=110 ;
1366:  !---------------------------- ;
1367:  !3By4 SR[1] INF, Max 36(Straight) ;
1368:  !R[103]=150 ;
1369:  !3By4 INF 45 Degree Diagonal Shif ;
1370:  !R[103]=160 ;
1371:  !---------------------------- ;
1372:  !R[103] "JOB_PROFILE" Selection ;
1373:  R[103]=150    ;
1374:  CALL JOB_VAR_COMMON(R[103]) ;
1375:   ;
1376:  ENDIF ;
1377:   ;
1378:  JMP LBL[9999] ;
1379:   ;
1380:  !Job 102681826 Logic Ends ;
1381:  !--------------------------- ;
1382:   ;
1383:  LBL[2047] ;
1384:  !--------------------------- ;
1385:  !Ring,Spacer ;
1386:  !Item 102772047 , Rev B ;
1387:  !Last Modified: 2022-04-14 ;
1388:  !Modified by: Tsuu ;
1389:  !0.5 IN Height ;
1390:  !1.54 IN ID, 3.96 IN OD ;
1391:  !ID Jaw # 1031 ;
1392:  !--------------------------- ;
1393:  IF (R[70]=2047) THEN ;
1394:   ;
1395:  !Define Parameters for INF/OTF ;
1396:  !R[105]=AR[1]=100, 2By3 Sheet ;
1397:  !R[105]=AR[1]=200, 3By4 Sheet ;
1398:  CALL JOB_VAR_SETUP(200) ;
1399:   ;
1400:  !--------------------------- ;
1401:  !Define Parameters for Job ;
1402:  !R[85] "INF_JAW_OFFSET"(Hgt) ;
1403:  R[85]=5    ;
1404:  !R[86] "INF_PICK_OFFSET" 50mm/sec ;
1405:  R[86]=1    ;
1406:  !R[87] "MAIN_LOAD_OFFSET" (PRELOA ;
1407:  R[87]=0    ;
1408:  !R[100] "GRIPPER_ID" 3 values ;
1409:  !If =100, ID Grippers Installed ;
1410:  !If =200, OD Grippers Installed ;
1411:  !If =300, OD 45 Degree Grippers ;
1412:  R[100]=100    ;
1413:  !--------------------------- ;
1414:   ;
1415:  !If using previous setup data ;
1416:  IF (R[71]=2047) THEN ;
1417:   ;
1418:  !--------------------------- ;
1419:  !1st: Height of Raw piece ;
1420:  R[190]=21.84    ;
1421:  !2nd: Height of Finish piece ;
1422:  R[191]=19.05    ;
1423:  !3rd: Infeed Height Offset ;
1424:  R[192]=(-4.5)    ;
1425:  !4th: Outfeed Height Offset ;
1426:  R[193]=(-53)    ;
1427:  !--------------------------- ;
1428:   ;
1429:  CALL CREATE_REG(R[190],R[191],R[192],R[193]) ;
1430:   ;
1431:  ENDIF ;
1432:   ;
1433:  !If new loading or offloading pos ;
1434:  !SET R[104] "IMPORT_LOADPOS" ;
1435:  !SET R[104]=1000, Otherwise NO ;
1436:  R[104]=1000    ;
1437:  IF (R[104]=1000) THEN ;
1438:  !R[260]=43, Preload Pos1 ;
1439:  !R[270]=44, Preload PosFinal ;
1440:  !R[300]=53, Offload PosFinal ;
1441:  !PR[43] Pre-Loading Pos1 ;
1442:  CALL CREATE_PR(43,169.843,(-60.088),270.324,20.863,88.464,19.016) ;
1443:  !PR[44] Final Loading Position ;
1444:  CALL CREATE_PR(44,169.552,(-60.299),282.077,20.856,88.465,19.003) ;
1445:  !PR[53] pre-Unloading Position ;
1446:  CALL CREATE_PR(53,(-131.864),93.832,251.814,171.263,(-88.238),(-173.098)) ;
1447:  !PR[54] Final Unloading Position ;
1448:  CALL CREATE_PR(54,(-131.564),93.953,241.127,171.244,(-88.239),(-173.082)) ;
1449:  !PR[56] assitant Unloading preses ;
1450:  CALL CREATE_PR(56,(-133.84),95.467,273.686,(-177.134),(-88.249),175.184) ;
1451:  !PR[57] assitant Unloading preses ;
1452:  CALL CREATE_PR(57,(-135.964),108.085,344.284,(-177.144),(-88.245),175.194) ;
1453:  !PR[58] assitant Unloading preses ;
1454:  CALL CREATE_PR(58,296.854,360.959,378.47,(-91.75),(-.28),88.063) ;
1455:  ENDIF ;
1456:   ;
1457:  !---------------------------- ;
1458:  !SR[1] = "JOB_VAR_ID_GRIP" ;
1459:  !JOB_VAR_COMMON(R[103])'s value ;
1460:  !---------------------------- ;
1461:  !2By3 SR[1] INF, Max 18(Straight) ;
1462:  !R[103]=100 ;
1463:  !2By3 INF 45 Degree Diagonal Shif ;
1464:  !R[103]=110 ;
1465:  !---------------------------- ;
1466:  !3By4 SR[1] INF, Max 36(Straight) ;
1467:  !R[103]=150 ;
1468:  !3By4 INF 45 Degree Diagonal Shif ;
1469:  !R[103]=160 ;
1470:  !---------------------------- ;
1471:  !R[103] "JOB_PROFILE" Selection ;
1472:  R[103]=150    ;
1473:  CALL JOB_VAR_COMMON(R[103]) ;
1474:   ;
1475:  ENDIF ;
1476:   ;
1477:  JMP LBL[9999] ;
1478:   ;
1479:  !Job 102772047 Logic Ends ;
1480:  !--------------------------- ;
1481:   ;
1482:  LBL[2052] ;
1483:  !--------------------------- ;
1484:  !Wedge ;
1485:  !Item 102772052 , Rev C ;
1486:  !Last Modified: 2022-12-20 ;
1487:  !Modified by: Tsuu ;
1488:  !2.53 IN Height ;
1489:  !2.02 IN ID, 3.75 IN OD ;
1490:  !ID Jaw # 1031 ;
1491:  !--------------------------- ;
1492:  IF (R[70]=2052) THEN ;
1493:   ;
1494:  !Define Parameters for INF/OTF ;
1495:  !R[105]=AR[1]=100, 2By3 Sheet ;
1496:  !R[105]=AR[1]=200, 3By4 Sheet ;
1497:  CALL JOB_VAR_SETUP(200) ;
1498:   ;
1499:  !--------------------------- ;
1500:  !Define Parameters for Job ;
1501:  !R[85] "INF_JAW_OFFSET"(Hgt) ;
1502:  R[85]=10    ;
1503:  !R[86] "INF_PICK_OFFSET" 50mm/sec ;
1504:  R[86]=1    ;
1505:  !R[87] "MAIN_LOAD_OFFSET" (PRELOA ;
1506:  R[87]=0    ;
1507:  !R[100] "GRIPPER_ID" 3 values ;
1508:  !If =100, ID Grippers Installed ;
1509:  !If =200, OD Grippers Installed ;
1510:  !If =300, OD 45 Degree Grippers ;
1511:  R[100]=100    ;
1512:  !--------------------------- ;
1513:   ;
1514:  !If using previous setup data ;
1515:  IF (R[71]=2052) THEN ;
1516:   ;
1517:  !--------------------------- ;
1518:  !1st: Height of Raw piece ;
1519:  R[190]=67    ;
1520:  !2nd: Height of Finish piece ;
1521:  R[191]=64.262    ;
1522:  !3rd: Infeed Height Offset ;
1523:  R[192]=(-5)    ;
1524:  !4th: Outfeed Height Offset ;
1525:  !Changing 1st Level Offset to ;
1526:  R[193]=(-21)    ;
1527:   ;
1528:  !Changing 2nd Level Offset to ;
1529:  R[194]=(-24)    ;
1530:   ;
1531:  !Changing 3rd Level Offset to ;
1532:  R[195]=(-27)    ;
1533:   ;
1534:  CALL GN_OUTFEED_COMPENSATE(R[193],R[194],R[195]) ;
1535:  !--------------------------- ;
1536:   ;
1537:  CALL CREATE_REG(R[190],R[191],R[192],R[193]) ;
1538:   ;
1539:  ENDIF ;
1540:   ;
1541:  !If new loading or offloading pos ;
1542:  !SET R[104] "IMPORT_LOADPOS" ;
1543:  !SET R[104]=1000, Otherwise NO ;
1544:  R[104]=1000    ;
1545:  IF (R[104]=1000) THEN ;
1546:  !R[260]=43, Preload Pos1 ;
1547:  !R[270]=44, Preload PosFinal ;
1548:  !R[300]=53, Offload PosFinal ;
1549:  !PR[43] Pre-Loading Pos1 ;
1550:  CALL CREATE_PR(43,168.636,(-60.568),289.828,29.541,89.225,27.754) ;
1551:  !PR[44] Final Loading Position ;
1552:  CALL CREATE_PR(44,168.542,(-60.702),299.286,29.558,89.226,27.768) ;
1553:  !PR[53] pre-Unloading Position ;
1554:  CALL CREATE_PR(53,(-127.956),94.46,95.432,172.755,(-88.217),(-174.592)) ;
1555:  !PR[54] Final Unloading Position ;
1556:  CALL CREATE_PR(54,(-126.861),94.652,59.692,172.766,(-88.216),(-174.606)) ;
1557:  !PR[56] assitant Unloading preses ;
1558:  CALL CREATE_PR(56,(-133.84),95.467,273.686,(-177.134),(-88.249),175.184) ;
1559:  !PR[57] assitant Unloading preses ;
1560:  CALL CREATE_PR(57,(-135.964),108.085,344.284,(-177.144),(-88.245),175.194) ;
1561:  !PR[58] assitant Unloading preses ;
1562:  CALL CREATE_PR(58,296.854,360.959,378.47,(-91.75),(-.28),88.063) ;
1563:  ENDIF ;
1564:   ;
1565:  !---------------------------- ;
1566:  !SR[1] = "JOB_VAR_ID_GRIP" ;
1567:  !JOB_VAR_COMMON(R[103])'s value ;
1568:  !---------------------------- ;
1569:  !2By3 SR[1] INF, Max 18(Straight) ;
1570:  !R[103]=100 ;
1571:  !2By3 INF 45 Degree Diagonal Shif ;
1572:  !R[103]=110 ;
1573:  !---------------------------- ;
1574:  !3By4 SR[1] INF, Max 36(Straight) ;
1575:  !R[103]=150 ;
1576:  !3By4 INF 45 Degree Diagonal Shif ;
1577:  !R[103]=160 ;
1578:  !---------------------------- ;
1579:  !R[103] "JOB_PROFILE" Selection ;
1580:  R[103]=150    ;
1581:  CALL JOB_VAR_COMMON(R[103]) ;
1582:   ;
1583:  ENDIF ;
1584:   ;
1585:  JMP LBL[9999] ;
1586:   ;
1587:  !Job 102772052 Logic Ends ;
1588:  !--------------------------- ;
1589:   ;
1590:  LBL[2126] ;
1591:  !--------------------------- ;
1592:  !Slip,Lower ;
1593:  !Item 103062126 , Rev A ;
1594:  !Last Modified: 2026-02-12 ;
1595:  !Modified by: Aaron ;
1596:  !4.00 IN Height ;
1597:  !3.94 IN ID, 5.86 IN OD, 32.0 Lbs ;
1598:  !ID Jaw # 1007 ;
1599:  !--------------------------- ;
1600:  IF (R[70]=2126) THEN ;
1601:   ;
1602:  !Define Parameters for INF/OTF ;
1603:  !R[105]=AR[1]=100, 2By3 Sheet ;
1604:  !R[105]=AR[1]=200, 3By4 Sheet ;
1605:  CALL JOB_VAR_SETUP(100) ;
1606:   ;
1607:  !--------------------------- ;
1608:  !Define Parameters for Job ;
1609:  R[1]=1    ;
1610:  R[2]=0    ;
1611:  R[4]=0    ;
1612:  R[67]=40    ;
1613:  !R[85] "INF_JAW_OFFSET"(Hgt) ;
1614:  R[85]=92.55    ;
1615:  !R[86] "INF_PICK_OFFSET" 50mm/sec ;
1616:  R[86]=0    ;
1617:  !R[87] "MAIN_LOAD_OFFSET" (PRELOA ;
1618:  R[87]=0    ;
1619:  !R[100] "GRIPPER_ID" 3 values ;
1620:  !If =100, ID Grippers Installed ;
1621:  !If =200, OD Grippers Installed ;
1622:  !If =300, OD 45 Degree Grippers ;
1623:  R[100]=100    ;
1624:  !--------------------------- ;
1625:   ;
1626:  !If using previous setup data ;
1627:  IF (R[71]=2126) THEN ;
1628:   ;
1629:  !--------------------------- ;
1630:  !1st: Height of Raw piece ;
1631:  R[190]=127.26    ;
1632:  !2nd: Height of Finish piece ;
1633:  R[191]=101.6    ;
1634:  !3rd: Infeed Height Offset ;
1635:  R[192]=(-285)    ;
1636:  !4th: Outfeed Height Offset ;
1637:  R[193]=(-235)    ;
1638:  !--------------------------- ;
1639:   ;
1640:  CALL CREATE_REG(R[190],R[191],R[192],R[193]) ;
1641:   ;
1642:  ENDIF ;
1643:   ;
1644:  !If new loading or offloading pos ;
1645:  !SET R[104] "IMPORT_LOADPOS" ;
1646:  !SET R[104]=1000, Otherwise NO ;
1647:  R[104]=1000    ;
1648:  IF (R[104]=1000) THEN ;
1649:  !R[260]=43, Preload Pos1 ;
1650:  !R[270]=44, Preload PosFinal ;
1651:  !R[300]=53, Offload PosFinal ;
1652:  !PR[43] Pre-Loading Pos1 ;
1653:  CALL CREATE_PR(43,167.386,(-64.099),283.406,154.866,89.247,153.365) ;
1654:  !PR[44] Final Loading Position ;
1655:  CALL CREATE_PR(44,167.746,(-64.039),315.752,155.332,89.254,153.845) ;
1656:  !PR[53] pre-Unloading Position ;
1657:  CALL CREATE_PR(53,(-130.325),93.623,168.029,168.855,(-88.276),(-170.226)) ;
1658:  !PR[54] Final Unloading Position ;
1659:  CALL CREATE_PR(54,(-128.735),93.392,117.767,169.08,(-88.268),(-170.429)) ;
1660:  !PR[56] assitant Unloading preses ;
1661:  CALL CREATE_PR(56,(-133.84),95.467,273.686,(-177.134),(-88.249),175.184) ;
1662:  !PR[57] assitant Unloading preses ;
1663:  CALL CREATE_PR(57,(-135.964),108.085,344.284,(-177.144),(-88.245),175.194) ;
1664:  !PR[58] assitant Unloading preses ;
1665:  CALL CREATE_PR(58,296.854,360.959,378.47,(-91.75),(-.28),88.063) ;
1666:  ENDIF ;
1667:   ;
1668:  !---------------------------- ;
1669:  !SR[1] = "JOB_VAR_ID_GRIP" ;
1670:  !JOB_VAR_COMMON(R[103])'s value ;
1671:  !---------------------------- ;
1672:  !2By3 SR[1] INF, Max 18(Straight) ;
1673:  !R[103]=100 ;
1674:  !2By3 INF 45 Degree Diagonal Shif ;
1675:  !R[103]=110 ;
1676:  !---------------------------- ;
1677:  !3By4 SR[1] INF, Max 36(Straight) ;
1678:  !R[103]=150 ;
1679:  !3By4 INF 45 Degree Diagonal Shif ;
1680:  !R[103]=160 ;
1681:  !---------------------------- ;
1682:  !R[103] "JOB_PROFILE" Selection ;
1683:  R[103]=100    ;
1684:  CALL JOB_VAR_COMMON(R[103]) ;
1685:   ;
1686:  ENDIF ;
1687:   ;
1688:  JMP LBL[9999] ;
1689:   ;
1690:  !Job 103062126 Logic Ends ;
1691:  !--------------------------- ;
1692:   ;
1693:  LBL[2407] ;
1694:  !--------------------------- ;
1695:  !Mandrel ;
1696:  !Item 102592407 , Rev B ;
1697:  !Last Modified: 2021-02-23 ;
1698:  !Modified by: Tsuu ;
1699:  !13.64 IN Height ;
1700:  !1.3 IN ID, 3.08 IN OD ;
1701:  !ID Jaw # Mandrel ;
1702:  !--------------------------- ;
1703:  IF (R[70]=2407) THEN ;
1704:   ;
1705:  !Define Parameters for INF/OTF ;
1706:  !R[105]=AR[1]=100, 2By3 Sheet ;
1707:  !R[105]=AR[1]=200, 3By4 Sheet ;
1708:  CALL JOB_VAR_SETUP(500) ;
1709:   ;
1710:  !--------------------------- ;
1711:  !Define Parameters for Job ;
1712:  !R[85] "INF_JAW_OFFSET"(Hgt) ;
1713:  R[85]=87.6    ;
1714:  !R[86] "INF_PICK_OFFSET" 50mm/sec ;
1715:  R[86]=20    ;
1716:  !R[87] "MAIN_LOAD_OFFSET" (PRELOA ;
1717:  R[87]=0    ;
1718:  !R[100] "GRIPPER_ID" 3 values ;
1719:  !If =100, ID Grippers Installed ;
1720:  !If =200, OD Grippers Installed ;
1721:  !If =300, OD 45 Degree Grippers ;
1722:  R[100]=100    ;
1723:  !--------------------------- ;
1724:   ;
1725:  !If using previous setup data ;
1726:  IF (R[71]=2407) THEN ;
1727:   ;
1728:  !--------------------------- ;
1729:  !1st: Height of Raw piece ;
1730:  R[190]=352    ;
1731:  !2nd: Height of Finish piece ;
1732:  R[191]=346.454    ;
1733:  !3rd: Infeed Height Offset ;
1734:  R[192]=(-69)    ;
1735:  !4th: Outfeed Height Offset ;
1736:  R[193]=(-167)    ;
1737:  !--------------------------- ;
1738:   ;
1739:  CALL CREATE_REG(R[190],R[191],R[192],R[193]) ;
1740:   ;
1741:  ENDIF ;
1742:   ;
1743:  !If new loading or offloading pos ;
1744:  !SET R[104] "IMPORT_LOADPOS" ;
1745:  !SET R[104]=1000, Otherwise NO ;
1746:  R[104]=1000    ;
1747:  IF (R[104]=1000) THEN ;
1748:  !R[260]=43, Preload Pos1 ;
1749:  !R[270]=44, Preload PosFinal ;
1750:  !R[300]=53, Offload PosFinal ;
1751:  !PR[43] Pre-Loading Pos1 ;
1752:  CALL CREATE_PR(43,167.549,(-70.776),(-18.955),149.368,88.995,147.238) ;
1753:  !PR[44] Final Loading Position ;
1754:  CALL CREATE_PR(44,169.813,(-71.016),130.131,149.353,88.991,147.2) ;
1755:  !PR[53] pre-Unloading Position ;
1756:  CALL CREATE_PR(53,(-132.181),108.408,216.873,173.351,(-88.246),(-175.317)) ;
1757:  !PR[54] Final Unloading Position ;
1758:  CALL CREATE_PR(54,(-127.063),108.782,47.825,173.531,(-88.25),(-175.496)) ;
1759:  !PR[56] assitant Unloading preses ;
1760:  CALL CREATE_PR(56,(-132.935),108.031,243.66,(-177.212),(-88.249),175.253) ;
1761:  !PR[57] assitant Unloading preses ;
1762:  CALL CREATE_PR(57,(-132.92),107.912,243.673,(-91.749),(-.28),88.057) ;
1763:  !PR[58] assitant Unloading preses ;
1764:  CALL CREATE_PR(58,296.854,360.959,378.47,(-91.75),(-.28),88.063) ;
1765:  ENDIF ;
1766:   ;
1767:  !---------------------------- ;
1768:  !SR[1] = "JOB_VAR_ID_GRIP" ;
1769:  !JOB_VAR_COMMON(R[103])'s value ;
1770:  !---------------------------- ;
1771:  !2By3 SR[1] INF, Max 18(Straight) ;
1772:  !R[103]=100 ;
1773:  !2By3 INF 45 Degree Diagonal Shif ;
1774:  !R[103]=110 ;
1775:  !---------------------------- ;
1776:  !3By4 SR[1] INF, Max 36(Straight) ;
1777:  !R[103]=150 ;
1778:  !3By4 INF 45 Degree Diagonal Shif ;
1779:  !R[103]=160 ;
1780:  !---------------------------- ;
1781:  !R[103] "JOB_PROFILE" Selection ;
1782:  R[103]=160    ;
1783:  CALL JOB_VAR_COMMON(R[103]) ;
1784:   ;
1785:  ENDIF ;
1786:   ;
1787:  JMP LBL[9999] ;
1788:   ;
1789:  !Job 102592407 Logic Ends ;
1790:  !--------------------------- ;
1791:   ;
1792:  !--------------------------- ;
1793:  LBL[2408] ;
1794:  !--------------------------- ;
1795:  !Ring,Spacer ;
1796:  !Item 102592408 , Rev C ;
1797:  !Last Modified: 2023-02-10 ;
1798:  !Modified by: Tsuu ;
1799:  !0.5 IN Height ;
1800:  !2.02 IN ID, 3.54 IN OD ;
1801:  !ID Jaw # 1031 ;
1802:  !--------------------------- ;
1803:  IF (R[70]=2408) THEN ;
1804:   ;
1805:  !Define Parameters for INF/OTF ;
1806:  !R[105]=AR[1]=100, 2By3 Sheet ;
1807:  !R[105]=AR[1]=200, 3By4 Sheet ;
1808:  CALL JOB_VAR_SETUP(200) ;
1809:   ;
1810:  !--------------------------- ;
1811:  !Define Parameters for Job ;
1812:  !R[85] "INF_JAW_OFFSET"(Hgt) ;
1813:  R[85]=5    ;
1814:  !R[86] "INF_PICK_OFFSET" 50mm/sec ;
1815:  R[86]=1    ;
1816:  !R[87] "MAIN_LOAD_OFFSET" (PRELOA ;
1817:  R[87]=0    ;
1818:  !R[100] "GRIPPER_ID" 3 values ;
1819:  !If =100, ID Grippers Installed ;
1820:  !If =200, OD Grippers Installed ;
1821:  !If =300, OD 45 Degree Grippers ;
1822:  R[100]=100    ;
1823:  !--------------------------- ;
1824:   ;
1825:  !If using previous setup data ;
1826:  IF (R[71]=2408) THEN ;
1827:   ;
1828:  !--------------------------- ;
1829:  !1st: Height of Raw piece ;
1830:  R[190]=15.62    ;
1831:  !2nd: Height of Finish piece ;
1832:  R[191]=12.7    ;
1833:  !3rd: Infeed Height Offset ;
1834:  R[192]=(-14)    ;
1835:  !4th: Outfeed Height Offset ;
1836:  R[193]=(-57)    ;
1837:  !--------------------------- ;
1838:   ;
1839:  CALL CREATE_REG(R[190],R[191],R[192],R[193]) ;
1840:   ;
1841:  ENDIF ;
1842:   ;
1843:  !If new loading or offloading pos ;
1844:  !SET R[104] "IMPORT_LOADPOS" ;
1845:  !SET R[104]=1000, Otherwise NO ;
1846:  R[104]=1000    ;
1847:  IF (R[104]=1000) THEN ;
1848:  !R[260]=43, Preload Pos1 ;
1849:  !R[270]=44, Preload PosFinal ;
1850:  !R[300]=53, Offload PosFinal ;
1851:  !PR[43] Pre-Loading Pos1 ;
1852:  CALL CREATE_PR(43,168.672,(-60.32),286.786,19.084,88.42,17.227) ;
1853:  !PR[44] Final Loading Position ;
1854:  CALL CREATE_PR(44,168.942,(-60.701),297.303,19.118,88.425,17.26) ;
1855:  !PR[53] pre-Unloading Position ;
1856:  CALL CREATE_PR(53,(-131.629),93.837,242.229,172.716,(-88.209),(-174.573)) ;
1857:  !PR[54] Final Unloading Position ;
1858:  CALL CREATE_PR(54,(-131.424),93.782,234.425,172.817,(-88.215),(-174.673)) ;
1859:  !PR[56] assitant Unloading preses ;
1860:  CALL CREATE_PR(56,(-133.84),95.467,273.686,(-177.134),(-88.249),175.184) ;
1861:  !PR[57] assitant Unloading preses ;
1862:  CALL CREATE_PR(57,(-135.964),108.085,344.284,(-177.144),(-88.245),175.194) ;
1863:  !PR[58] assitant Unloading preses ;
1864:  CALL CREATE_PR(58,296.854,360.959,378.47,(-91.75),(-.28),88.063) ;
1865:  ENDIF ;
1866:   ;
1867:  !---------------------------- ;
1868:  !SR[1] = "JOB_VAR_ID_GRIP" ;
1869:  !JOB_VAR_COMMON(R[103])'s value ;
1870:  !---------------------------- ;
1871:  !2By3 SR[1] INF, Max 18(Straight) ;
1872:  !R[103]=100 ;
1873:  !2By3 INF 45 Degree Diagonal Shif ;
1874:  !R[103]=110 ;
1875:  !---------------------------- ;
1876:  !3By4 SR[1] INF, Max 36(Straight) ;
1877:  !R[103]=150 ;
1878:  !3By4 INF 45 Degree Diagonal Shif ;
1879:  !R[103]=160 ;
1880:  !---------------------------- ;
1881:  !R[103] "JOB_PROFILE" Selection ;
1882:  R[103]=150    ;
1883:  CALL JOB_VAR_COMMON(R[103]) ;
1884:   ;
1885:  ENDIF ;
1886:   ;
1887:  JMP LBL[9999] ;
1888:   ;
1889:  !Job 102592408 Logic Ends ;
1890:  !--------------------------- ;
1891:   ;
1892:  !--------------------------- ;
1893:  LBL[3245] ;
1894:  !--------------------------- ;
1895:  !Retainer, Lower ;
1896:  !Item 101463245 , Rev A ;
1897:  !Last Modified: 2026-01-25 ;
1898:  !Modified by: Aaron ;
1899:  !1.49 IN Height ;
1900:  !5.59 IN ID, 5.9 IN OD, 7.0 Lbs W ;
1901:  !ID Jaw # 1004 ;
1902:  !--------------------------- ;
1903:  IF (R[70]=3245) THEN ;
1904:   ;
1905:  !Define Parameters for INF/OTF ;
1906:  !R[105]=AR[1]=100, 2By3 Sheet ;
1907:  !R[105]=AR[1]=200, 3By4 Sheet ;
1908:  CALL JOB_VAR_SETUP(100) ;
1909:   ;
1910:  !--------------------------- ;
1911:  !Define Parameters for Job ;
1912:  R[1]=1    ;
1913:  R[2]=0    ;
1914:  R[4]=0    ;
1915:  R[67]=20    ;
1916:  !R[85] "INF_JAW_OFFSET"(Hgt) ;
1917:  R[85]=20    ;
1918:  !R[86] "INF_PICK_OFFSET" 50mm/sec ;
1919:  R[86]=2    ;
1920:  !R[87] "MAIN_LOAD_OFFSET" (PRELOA ;
1921:  R[87]=0    ;
1922:  !R[100] "GRIPPER_ID" 3 values ;
1923:  !If =100, ID Grippers Installed ;
1924:  !If =200, OD Grippers Installed ;
1925:  !If =300, OD 45 Degree Grippers ;
1926:  R[100]=100    ;
1927:  !--------------------------- ;
1928:   ;
1929:  !If using previous setup data ;
1930:  IF (R[71]=3245) THEN ;
1931:   ;
1932:  !--------------------------- ;
1933:  !1st: Height of Raw piece ;
1934:  R[190]=31.37    ;
1935:  !2nd: Height of Finish piece ;
1936:  R[191]=25.27    ;
1937:  !3rd: Infeed Height Offset ;
1938:  R[192]=(-255)    ;
1939:  !4th: Outfeed Height Offset ;
1940:  R[193]=(-300)    ;
1941:  !--------------------------- ;
1942:   ;
1943:  CALL CREATE_REG(R[190],R[191],R[192],R[193]) ;
1944:   ;
1945:  ENDIF ;
1946:   ;
1947:  !If new loading or offloading pos ;
1948:  !SET R[104] "IMPORT_LOADPOS" ;
1949:  !SET R[104]=1000, Otherwise NO ;
1950:  R[104]=1000    ;
1951:  IF (R[104]=1000) THEN ;
1952:  !R[260]=43, Preload Pos1 ;
1953:  !R[270]=44, Preload PosFinal ;
1954:  !R[300]=53, Offload PosFinal ;
1955:  !PR[43] Pre-Loading Pos1 ;
1956:  CALL CREATE_PR(43,168.298,(-62.409),352.328,(-149.037),88.885,(-150.921)) ;
1957:  !PR[44] Final Loading Position ;
1958:  CALL CREATE_PR(44,168.733,(-62.054),375.302,(-149.343),88.879,(-151.222)) ;
1959:  !PR[53] pre-Unloading Position ;
1960:  CALL CREATE_PR(53,(-126.862),94.747,73.49,172.899,(-88.227),(-174.493)) ;
1961:  !PR[54] Final Unloading Position ;
1962:  CALL CREATE_PR(54,(-126.241),95.015,51.542,172.164,(-88.238),(-173.761)) ;
1963:  !PR[56] assitant Unloading preses ;
1964:  CALL CREATE_PR(56,(-133.84),95.467,273.686,(-177.134),(-88.249),175.184) ;
1965:  !PR[57] assitant Unloading preses ;
1966:  CALL CREATE_PR(57,(-135.964),108.085,344.284,(-177.144),(-88.245),175.194) ;
1967:  !PR[58] assitant Unloading preses ;
1968:  CALL CREATE_PR(58,296.854,360.959,378.47,(-91.75),(-.28),88.063) ;
1969:  ENDIF ;
1970:   ;
1971:  !---------------------------- ;
1972:  !SR[1] = "JOB_VAR_ID_GRIP" ;
1973:  !JOB_VAR_COMMON(R[103])'s value ;
1974:  !---------------------------- ;
1975:  !2By3 SR[1] INF, Max 18(Straight) ;
1976:  !R[103]=100 ;
1977:  !2By3 INF 45 Degree Diagonal Shif ;
1978:  !R[103]=110 ;
1979:  !---------------------------- ;
1980:  !3By4 SR[1] INF, Max 36(Straight) ;
1981:  !R[103]=150 ;
1982:  !3By4 INF 45 Degree Diagonal Shif ;
1983:  !R[103]=160 ;
1984:  !---------------------------- ;
1985:  !R[103] "JOB_PROFILE" Selection ;
1986:  R[103]=100    ;
1987:  CALL JOB_VAR_COMMON(R[103]) ;
1988:   ;
1989:  ENDIF ;
1990:   ;
1991:  JMP LBL[9999] ;
1992:   ;
1993:  !Job 101463245 Logic Ends ;
1994:  !--------------------------- ;
1995:   ;
1996:  LBL[3284] ;
1997:  !--------------------------- ;
1998:  !Wedge ;
1999:  !Item 102503284 , Rev C ;
2000:  !Last Modified: 2023-02-21 ;
2001:  !Modified by: Tsuu ;
2002:  !2.16 IN Height ;
2003:  !2.01 IN ID, 3.46 IN OD ;
2004:  !ID Jaw # 1031 ;
2005:  !--------------------------- ;
2006:  IF (R[70]=3284) THEN ;
2007:   ;
2008:  !Define Parameters for INF/OTF ;
2009:  !R[105]=AR[1]=100, 2By3 Sheet ;
2010:  !R[105]=AR[1]=200, 3By4 Sheet ;
2011:  CALL JOB_VAR_SETUP(200) ;
2012:   ;
2013:  !--------------------------- ;
2014:  !Define Parameters for Job ;
2015:  !R[85] "INF_JAW_OFFSET"(Hgt) ;
2016:  R[85]=10    ;
2017:  !R[86] "INF_PICK_OFFSET" 50mm/sec ;
2018:  R[86]=5    ;
2019:  !R[87] "MAIN_LOAD_OFFSET" (PRELOA ;
2020:  R[87]=0    ;
2021:  !R[100] "GRIPPER_ID" 3 values ;
2022:  !If =100, ID Grippers Installed ;
2023:  !If =200, OD Grippers Installed ;
2024:  !If =300, OD 45 Degree Grippers ;
2025:  R[100]=100    ;
2026:  !--------------------------- ;
2027:   ;
2028:  !If using previous setup data ;
2029:  IF (R[71]=3284) THEN ;
2030:   ;
2031:  !--------------------------- ;
2032:  !1st: Height of Raw piece ;
2033:  R[190]=57.404    ;
2034:  !2nd: Height of Finish piece ;
2035:  R[191]=54.864    ;
2036:  !3rd: Infeed Height Offset ;
2037:  R[192]=(-13)    ;
2038:  !4th: Outfeed Height Offset ;
2039:  !Changing 1st Level Offset to ;
2040:  R[193]=(-32)    ;
2041:   ;
2042:  !Changing 2nd Level Offset to ;
2043:  R[194]=(-35)    ;
2044:   ;
2045:  !Changing 3rd Level Offset to ;
2046:  R[195]=(-38)    ;
2047:   ;
2048:  CALL GN_OUTFEED_COMPENSATE(R[193],R[194],R[195]) ;
2049:  !--------------------------- ;
2050:   ;
2051:  CALL CREATE_REG(R[190],R[191],R[192],R[193]) ;
2052:   ;
2053:  ENDIF ;
2054:   ;
2055:  !If new loading or offloading pos ;
2056:  !SET R[104] "IMPORT_LOADPOS" ;
2057:  !SET R[104]=1000, Otherwise NO ;
2058:  R[104]=1000    ;
2059:  IF (R[104]=1000) THEN ;
2060:  !R[260]=43, Preload Pos1 ;
2061:  !R[270]=44, Preload PosFinal ;
2062:  !R[300]=53, Offload PosFinal ;
2063:  !PR[43] Pre-Loading Pos1 ;
2064:  CALL CREATE_PR(43,168.498,(-59.875),303.928,39.992,88.975,38.229) ;
2065:  !PR[44] Final Loading Position ;
2066:  CALL CREATE_PR(44,168.332,(-60.115),317.433,40.065,88.977,38.298) ;
2067:  !PR[53] pre-Unloading Position ;
2068:  CALL CREATE_PR(53,(-127.251),94.418,83.107,166.328,(-88.32),(-168.136)) ;
2069:  !PR[54] Final Unloading Position ;
2070:  CALL CREATE_PR(54,(-126.424),94.659,54.252,166.39,(-88.319),(-168.2)) ;
2071:  !PR[56] assitant Unloading preses ;
2072:  CALL CREATE_PR(56,(-133.84),95.467,273.686,(-177.134),(-88.249),175.184) ;
2073:  !PR[57] assitant Unloading preses ;
2074:  CALL CREATE_PR(57,(-135.964),108.085,344.284,(-177.144),(-88.245),175.194) ;
2075:  !PR[58] assitant Unloading preses ;
2076:  CALL CREATE_PR(58,296.854,360.959,378.47,(-91.75),(-.28),88.063) ;
2077:  ENDIF ;
2078:   ;
2079:  !---------------------------- ;
2080:  !SR[1] = "JOB_VAR_ID_GRIP" ;
2081:  !JOB_VAR_COMMON(R[103])'s value ;
2082:  !---------------------------- ;
2083:  !2By3 SR[1] INF, Max 18(Straight) ;
2084:  !R[103]=100 ;
2085:  !2By3 INF 45 Degree Diagonal Shif ;
2086:  !R[103]=110 ;
2087:  !---------------------------- ;
2088:  !3By4 SR[1] INF, Max 36(Straight) ;
2089:  !R[103]=150 ;
2090:  !3By4 INF 45 Degree Diagonal Shif ;
2091:  !R[103]=160 ;
2092:  !---------------------------- ;
2093:  !R[103] "JOB_PROFILE" Selection ;
2094:  R[103]=150    ;
2095:  CALL JOB_VAR_COMMON(R[103]) ;
2096:   ;
2097:  ENDIF ;
2098:   ;
2099:  JMP LBL[9999] ;
2100:   ;
2101:  !Job 102503284 Logic Ends ;
2102:  !--------------------------- ;
2103:   ;
2104:  LBL[3721] ;
2105:  !--------------------------- ;
2106:  !Slip ;
2107:  !Item 102703721 , Rev C ;
2108:  !Last Modified: 2023-01-27 ;
2109:  !Modified by: Tsuu ;
2110:  !1.92 IN Height ;
2111:  !3.16 IN ID, 4.760 IN OD ;
2112:  !ID Jaw # 1025 ;
2113:  !--------------------------- ;
2114:  IF (R[70]=3721) THEN ;
2115:   ;
2116:  !Define Parameters for INF/OTF ;
2117:  !R[105]=AR[1]=100, 2By3 Sheet ;
2118:  !R[105]=AR[1]=200, 3By4 Sheet ;
2119:  CALL JOB_VAR_SETUP(200) ;
2120:   ;
2121:  !--------------------------- ;
2122:  !Define Parameters for Job ;
2123:  !R[85] "INF_JAW_OFFSET"(Hgt) ;
2124:  R[85]=25    ;
2125:  !R[86] "INF_PICK_OFFSET" 50mm/sec ;
2126:  R[86]=13    ;
2127:  !R[87] "MAIN_LOAD_OFFSET" (PRELOA ;
2128:  R[87]=0    ;
2129:  !R[100] "GRIPPER_ID" 3 values ;
2130:  !If =100, ID Grippers Installed ;
2131:  !If =200, OD Grippers Installed ;
2132:  !If =300, OD 45 Degree Grippers ;
2133:  R[100]=100    ;
2134:  !--------------------------- ;
2135:   ;
2136:  !If using previous setup data ;
2137:  IF (R[71]=3721) THEN ;
2138:   ;
2139:  !--------------------------- ;
2140:  !1st: Height of Raw piece ;
2141:  R[190]=51.47    ;
2142:  !2nd: Height of Finish piece ;
2143:  R[191]=48.768    ;
2144:  !3rd: Infeed Height Offset ;
2145:  R[192]=(-52)    ;
2146:  !4th: Outfeed Height Offset ;
2147:  R[193]=(-90)    ;
2148:  !--------------------------- ;
2149:   ;
2150:  CALL CREATE_REG(R[190],R[191],R[192],R[193]) ;
2151:   ;
2152:  ENDIF ;
2153:   ;
2154:  !If new loading or offloading pos ;
2155:  !SET R[104] "IMPORT_LOADPOS" ;
2156:  !SET R[104]=1000, Otherwise NO ;
2157:  R[104]=1000    ;
2158:  IF (R[104]=1000) THEN ;
2159:  !R[260]=43, Preload Pos1 ;
2160:  !R[270]=44, Preload PosFinal ;
2161:  !R[300]=53, Offload PosFinal ;
2162:  !PR[43] Pre-Loading Pos1 ;
2163:  CALL CREATE_PR(43,169.345,(-60.542),354.26,67.682,89.47,65.865) ;
2164:  !PR[44] Final Loading Position ;
2165:  CALL CREATE_PR(44,169.317,(-60.748),365.389,67.731,89.47,65.911) ;
2166:  !PR[53] pre-Unloading Position ;
2167:  CALL CREATE_PR(53,(-125.093),95.886,36.656,173.09,(-88.208),(-174.916)) ;
2168:  !PR[54] Final Unloading Position ;
2169:  CALL CREATE_PR(54,(-123.627),95.762,(-9.141),173.225,(-88.208),(-175.035)) ;
2170:  !PR[56] assitant Unloading preses ;
2171:  CALL CREATE_PR(56,(-133.84),95.467,273.686,(-177.134),(-88.249),175.184) ;
2172:  !PR[57] assitant Unloading preses ;
2173:  CALL CREATE_PR(57,(-135.964),108.085,344.284,(-177.144),(-88.245),175.194) ;
2174:  !PR[58] assitant Unloading preses ;
2175:  CALL CREATE_PR(58,296.854,360.959,378.47,(-91.75),(-.28),88.063) ;
2176:  ENDIF ;
2177:   ;
2178:  !---------------------------- ;
2179:  !SR[1] = "JOB_VAR_ID_GRIP" ;
2180:  !JOB_VAR_COMMON(R[103])'s value ;
2181:  !---------------------------- ;
2182:  !2By3 SR[1] INF, Max 18(Straight) ;
2183:  !R[103]=100 ;
2184:  !2By3 INF 45 Degree Diagonal Shif ;
2185:  !R[103]=110 ;
2186:  !---------------------------- ;
2187:  !3By4 SR[1] INF, Max 36(Straight) ;
2188:  !R[103]=150 ;
2189:  !3By4 INF 45 Degree Diagonal Shif ;
2190:  !R[103]=160 ;
2191:  !---------------------------- ;
2192:  !R[103] "JOB_PROFILE" Selection ;
2193:  R[103]=150    ;
2194:  CALL JOB_VAR_COMMON(R[103]) ;
2195:   ;
2196:  ENDIF ;
2197:   ;
2198:  JMP LBL[9999] ;
2199:   ;
2200:  !Job 102703721 Logic Ends ;
2201:  !--------------------------- ;
2202:   ;
2203:  LBL[5613] ;
2204:  !--------------------------- ;
2205:  !Wedge ;
2206:  !Item 102745613 , Rev C ;
2207:  !Last Modified: 2023-03-01 ;
2208:  !Modified by: Tsuu ;
2209:  !2.40 IN Height ;
2210:  !2.01 IN ID, 3.46 IN OD ;
2211:  !ID Jaw # 1031 ;
2212:  !--------------------------- ;
2213:  IF (R[70]=5613) THEN ;
2214:   ;
2215:  !Define Parameters for INF/OTF ;
2216:  !R[105]=AR[1]=100, 2By3 Sheet ;
2217:  !R[105]=AR[1]=200, 3By4 Sheet ;
2218:  CALL JOB_VAR_SETUP(200) ;
2219:   ;
2220:  !--------------------------- ;
2221:  !Define Parameters for Job ;
2222:  !R[85] "INF_JAW_OFFSET"(Hgt) ;
2223:  R[85]=10    ;
2224:  !R[86] "INF_PICK_OFFSET" 50mm/sec ;
2225:  R[86]=5    ;
2226:  !R[87] "MAIN_LOAD_OFFSET" (PRELOA ;
2227:  R[87]=0    ;
2228:  !R[100] "GRIPPER_ID" 3 values ;
2229:  !If =100, ID Grippers Installed ;
2230:  !If =200, OD Grippers Installed ;
2231:  !If =300, OD 45 Degree Grippers ;
2232:  R[100]=100    ;
2233:  !--------------------------- ;
2234:   ;
2235:  !If using previous setup data ;
2236:  IF (R[71]=5613) THEN ;
2237:   ;
2238:  !--------------------------- ;
2239:  !1st: Height of Raw piece ;
2240:  R[190]=63.5    ;
2241:  !2nd: Height of Finish piece ;
2242:  R[191]=60.96    ;
2243:  !3rd: Infeed Height Offset ;
2244:  R[192]=(-13)    ;
2245:  !4th: Outfeed Height Offset ;
2246:  !Changing 1st Level Offset to ;
2247:  R[193]=(-26)    ;
2248:   ;
2249:  !Changing 2nd Level Offset to ;
2250:  R[194]=(-26)    ;
2251:   ;
2252:  !Changing 3rd Level Offset to ;
2253:  R[195]=(-26)    ;
2254:   ;
2255:  CALL GN_OUTFEED_COMPENSATE(R[193],R[194],R[195]) ;
2256:  !--------------------------- ;
2257:   ;
2258:  CALL CREATE_REG(R[190],R[191],R[192],R[193]) ;
2259:   ;
2260:  ENDIF ;
2261:   ;
2262:  !If new loading or offloading pos ;
2263:  !SET R[104] "IMPORT_LOADPOS" ;
2264:  !SET R[104]=1000, Otherwise NO ;
2265:  R[104]=1000    ;
2266:  IF (R[104]=1000) THEN ;
2267:  !R[260]=43, Preload Pos1 ;
2268:  !R[270]=44, Preload PosFinal ;
2269:  !R[300]=53, Offload PosFinal ;
2270:  !PR[43] Pre-Loading Pos1 ;
2271:  CALL CREATE_PR(43,168.34,(-59.237),294.359,129.783,89.102,128.057) ;
2272:  !PR[44] Final Loading Position ;
2273:  CALL CREATE_PR(44,168.503,(-59.508),309.049,129.895,89.101,128.164) ;
2274:  !PR[53] pre-Unloading Position ;
2275:  CALL CREATE_PR(53,(-127.892),94.224,101.759,162.89,(-88.35),(-164.668)) ;
2276:  !PR[54] Final Unloading Position ;
2277:  CALL CREATE_PR(54,(-126.656),94.628,56.811,162.912,(-88.351),(-164.695)) ;
2278:  !PR[56] assitant Unloading preses ;
2279:  CALL CREATE_PR(56,(-133.84),95.467,273.686,(-177.134),(-88.249),175.184) ;
2280:  !PR[57] assitant Unloading preses ;
2281:  CALL CREATE_PR(57,(-135.964),108.085,344.284,(-177.144),(-88.245),175.194) ;
2282:  !PR[58] assitant Unloading preses ;
2283:  CALL CREATE_PR(58,296.854,360.959,378.47,(-91.75),(-.28),88.063) ;
2284:  ENDIF ;
2285:   ;
2286:  !---------------------------- ;
2287:  !SR[1] = "JOB_VAR_ID_GRIP" ;
2288:  !JOB_VAR_COMMON(R[103])'s value ;
2289:  !---------------------------- ;
2290:  !2By3 SR[1] INF, Max 18(Straight) ;
2291:  !R[103]=100 ;
2292:  !2By3 INF 45 Degree Diagonal Shif ;
2293:  !R[103]=110 ;
2294:  !---------------------------- ;
2295:  !3By4 SR[1] INF, Max 36(Straight) ;
2296:  !R[103]=150 ;
2297:  !3By4 INF 45 Degree Diagonal Shif ;
2298:  !R[103]=160 ;
2299:  !---------------------------- ;
2300:  !R[103] "JOB_PROFILE" Selection ;
2301:  R[103]=150    ;
2302:  CALL JOB_VAR_COMMON(R[103]) ;
2303:   ;
2304:  ENDIF ;
2305:   ;
2306:  JMP LBL[9999] ;
2307:   ;
2308:  !Job 102745613 Logic Ends ;
2309:  !--------------------------- ;
2310:   ;
2311:  LBL[5791] ;
2312:  !--------------------------- ;
2313:  !Retainer, Element ;
2314:  !Item 103205791 , Rev A ;
2315:  !Last Modified: 2026-02-05 ;
2316:  !Modified by: Aaron ;
2317:  !1.55 IN Height ;
2318:  !4.56 IN ID, 5.75 IN OD, 7.5 Lbs ;
2319:  !ID Jaw # 1014 ;
2320:  !--------------------------- ;
2321:  IF (R[70]=5791) THEN ;
2322:   ;
2323:  !Define Parameters for INF/OTF ;
2324:  !R[105]=AR[1]=100, 2By3 Sheet ;
2325:  !R[105]=AR[1]=200, 3By4 Sheet ;
2326:  CALL JOB_VAR_SETUP(100) ;
2327:   ;
2328:  !--------------------------- ;
2329:  !Define Parameters for Job ;
2330:  R[1]=1    ;
2331:  R[2]=0    ;
2332:  R[4]=0    ;
2333:  R[67]=40    ;
2334:  !R[85] "INF_JAW_OFFSET"(Hgt) ;
2335:  R[85]=73.93    ;
2336:  !R[86] "INF_PICK_OFFSET" 50mm/sec ;
2337:  R[86]=0    ;
2338:  !R[87] "MAIN_LOAD_OFFSET" (PRELOA ;
2339:  R[87]=0    ;
2340:  !R[100] "GRIPPER_ID" 3 values ;
2341:  !If =100, ID Grippers Installed ;
2342:  !If =200, OD Grippers Installed ;
2343:  !If =300, OD 45 Degree Grippers ;
2344:  R[100]=100    ;
2345:  !--------------------------- ;
2346:   ;
2347:  !If using previous setup data ;
2348:  IF (R[71]=5791) THEN ;
2349:   ;
2350:  !--------------------------- ;
2351:  !1st: Height of Raw piece ;
2352:  R[190]=46.1    ;
2353:  !2nd: Height of Finish piece ;
2354:  R[191]=39.37    ;
2355:  !3rd: Infeed Height Offset ;
2356:  R[192]=(-295)    ;
2357:  !4th: Outfeed Height Offset ;
2358:  R[193]=(-320)    ;
2359:  !--------------------------- ;
2360:   ;
2361:  CALL CREATE_REG(R[190],R[191],R[192],R[193]) ;
2362:   ;
2363:  ENDIF ;
2364:   ;
2365:  !If new loading or offloading pos ;
2366:  !SET R[104] "IMPORT_LOADPOS" ;
2367:  !SET R[104]=1000, Otherwise NO ;
2368:  R[104]=1000    ;
2369:  IF (R[104]=1000) THEN ;
2370:  !R[260]=43, Preload Pos1 ;
2371:  !R[270]=44, Preload PosFinal ;
2372:  !R[300]=53, Offload PosFinal ;
2373:  !PR[43] Pre-Loading Pos1 ;
2374:  CALL CREATE_PR(43,167.634,(-61.21),332.868,125.606,88.913,123.74) ;
2375:  !PR[44] Final Loading Position ;
2376:  CALL CREATE_PR(44,168.397,(-62.456),330.583,(-139.386),87.88,(-141.147)) ;
2377:  !PR[53] pre-Unloading Position ;
2378:  CALL CREATE_PR(53,(-126.862),94.747,73.49,172.899,(-88.227),(-174.493)) ;
2379:  !PR[54] Final Unloading Position ;
2380:  CALL CREATE_PR(54,(-126.241),95.015,51.542,172.164,(-88.238),(-173.761)) ;
2381:  !PR[56] assitant Unloading preses ;
2382:  CALL CREATE_PR(56,(-133.84),95.467,273.686,(-177.134),(-88.249),175.184) ;
2383:  !PR[57] assitant Unloading preses ;
2384:  CALL CREATE_PR(57,(-135.964),108.085,344.284,(-177.144),(-88.245),175.194) ;
2385:  !PR[58] assitant Unloading preses ;
2386:  CALL CREATE_PR(58,296.854,360.959,378.47,(-91.75),(-.28),88.063) ;
2387:  ENDIF ;
2388:   ;
2389:  !---------------------------- ;
2390:  !SR[1] = "JOB_VAR_ID_GRIP" ;
2391:  !JOB_VAR_COMMON(R[103])'s value ;
2392:  !---------------------------- ;
2393:  !2By3 SR[1] INF, Max 18(Straight) ;
2394:  !R[103]=100 ;
2395:  !2By3 INF 45 Degree Diagonal Shif ;
2396:  !R[103]=110 ;
2397:  !---------------------------- ;
2398:  !3By4 SR[1] INF, Max 36(Straight) ;
2399:  !R[103]=150 ;
2400:  !3By4 INF 45 Degree Diagonal Shif ;
2401:  !R[103]=160 ;
2402:  !---------------------------- ;
2403:  !R[103] "JOB_PROFILE" Selection ;
2404:  R[103]=100    ;
2405:  CALL JOB_VAR_COMMON(R[103]) ;
2406:   ;
2407:  ENDIF ;
2408:   ;
2409:  JMP LBL[9999] ;
2410:   ;
2411:  !Job 103205791 Logic Ends ;
2412:  !--------------------------- ;
2413:   ;
2414:  LBL[6970] ;
2415:  !--------------------------- ;
2416:  !Weld ;
2417:  !Item 100006970 , Rev B ;
2418:  !Last Modified: 2026-04-27 ;
2419:  !Modified by: Aaron ;
2420:  !10.545 IN Height ;
2421:  !3.17 IN ID, 4.370 IN OD ;
2422:  !ID Jaw # 1013 ;
2423:  !--------------------------- ;
2424:  IF (R[70]=6970) THEN ;
2425:   ;
2426:  !Define Parameters for INF/OTF ;
2427:  !R[105]=AR[1]=100, 2By3 Sheet ;
2428:  !R[105]=AR[1]=200, 3By4 Sheet ;
2429:  CALL JOB_VAR_SETUP(100) ;
2430:   ;
2431:  !--------------------------- ;
2432:  !Define Parameters for Job ;
2433:  R[1]=1    ;
2434:  R[2]=1    ;
2435:  R[4]=1    ;
2436:  R[67]=100    ;
2437:  !R[85] "INF_JAW_OFFSET"(Hgt) ;
2438:  R[85]=165.77    ;
2439:  !R[86] "INF_PICK_OFFSET" 50mm/sec ;
2440:  R[86]=10    ;
2441:  !R[87] "MAIN_LOAD_OFFSET" (PRELOA ;
2442:  R[87]=0    ;
2443:  !R[100] "GRIPPER_ID" 3 values ;
2444:  !If =100, ID Grippers Installed ;
2445:  !If =200, OD Grippers Installed ;
2446:  !If =300, OD 45 Degree Grippers ;
2447:  R[100]=100    ;
2448:  !--------------------------- ;
2449:   ;
2450:  !If using previous setup data ;
2451:  IF (R[71]=6970) THEN ;
2452:   ;
2453:  !--------------------------- ;
2454:  !1st: Height of Raw piece ;
2455:  R[190]=267.842    ;
2456:  !2nd: Height of Finish piece ;
2457:  R[191]=250    ;
2458:  !3rd: Infeed Height Offset ;
2459:  R[192]=(-300)    ;
2460:  !4th: Outfeed Height Offset ;
2461:  R[193]=(-40)    ;
2462:  !--------------------------- ;
2463:   ;
2464:  CALL CREATE_REG(R[190],R[191],R[192],R[193]) ;
2465:   ;
2466:  ENDIF ;
2467:   ;
2468:  !If new loading or offloading pos ;
2469:  !SET R[104] "IMPORT_LOADPOS" ;
2470:  !SET R[104]=1000, Otherwise NO ;
2471:  R[104]=1000    ;
2472:  IF (R[104]=1000) THEN ;
2473:  !R[260]=43, Preload Pos1 ;
2474:  !R[270]=44, Preload PosFinal ;
2475:  !R[300]=53, Offload PosFinal ;
2476:  !PR[43] Pre-Loading Pos1 ;
2477:  CALL CREATE_PR(43,167.537,(-62.622),133.47,103.2,89.276,102.077) ;
2478:  !PR[44] Final Loading Position ;
2479:  CALL CREATE_PR(44,167.72,(-63.542),190.442,103.416,89.263,102.281) ;
2480:  !PR[53] pre-Unloading Position ;
2481:  CALL CREATE_PR(53,(-129.189),92.632,169.217,170.145,(-88.272),(-171.356)) ;
2482:  !PR[54] Final Unloading Position ;
2483:  CALL CREATE_PR(54,(-126.007),92.8665,62.07,170.397,(-88.274),(-171.597)) ;
2484:  !PR[56] assitant Unloading preses ;
2485:  CALL CREATE_PR(56,(-133.84),95.467,273.686,(-177.134),(-88.249),175.184) ;
2486:  !PR[57] assitant Unloading preses ;
2487:  CALL CREATE_PR(57,(-135.964),108.085,344.284,(-177.144),(-88.245),175.194) ;
2488:  !PR[58] assitant Unloading preses ;
2489:  CALL CREATE_PR(58,296.854,360.959,378.47,(-91.75),(-.28),88.063) ;
2490:  ENDIF ;
2491:   ;
2492:  !---------------------------- ;
2493:  !SR[1] = "JOB_VAR_ID_GRIP" ;
2494:  !JOB_VAR_COMMON(R[103])'s value ;
2495:  !---------------------------- ;
2496:  !2By3 SR[1] INF, Max 18(Straight) ;
2497:  !R[103]=100 ;
2498:  !2By3 INF 45 Degree Diagonal Shif ;
2499:  !R[103]=110 ;
2500:  !---------------------------- ;
2501:  !3By4 SR[1] INF, Max 36(Straight) ;
2502:  !R[103]=150 ;
2503:  !3By4 INF 45 Degree Diagonal Shif ;
2504:  !R[103]=160 ;
2505:  !---------------------------- ;
2506:  !R[103] "JOB_PROFILE" Selection ;
2507:  R[103]=100    ;
2508:  CALL JOB_VAR_COMMON(R[103]) ;
2509:   ;
2510:  ENDIF ;
2511:   ;
2512:  JMP LBL[9999] ;
2513:   ;
2514:  !Job 100006970 Logic Ends ;
2515:  !--------------------------- ;
2516:   ;
2517:  LBL[4857] ;
2518:  !--------------------------- ;
2519:  !Weld ;
2520:  !Item 101444857 , Rev A ;
2521:  !Last Modified: 2026-July-17 ;
2522:  !Modified by: Erfan ;
2523:  !4.5 IN Height ;
2524:  !3.25 IN ID, 4.5 IN OD ;
2525:  !ID Jaw # 1004 ;
2526:  !--------------------------- ;
2527:  IF (R[70]=4857) THEN ;
2528:   ;
2529:  !Define Parameters for INF/OTF ;
2530:  !R[105]=AR[1]=100, 2By3 Sheet ;
2531:  !R[105]=AR[1]=200, 3By4 Sheet ;
2532:  CALL JOB_VAR_SETUP(100) ;
2533:   ;
2534:  !--------------------------- ;
2535:  !Define Parameters for Job ;
2536:  R[1]=1    ;
2537:  R[2]=1    ;
2538:  R[4]=1    ;
2539:  R[67]=100    ;
2540:  !R[85] "INF_JAW_OFFSET"(Hgt) ;
2541:  R[85]=105    ;
2542:  !R[86] "INF_PICK_OFFSET" 50mm/sec ;
2543:  R[86]=10    ;
2544:  !R[87] "MAIN_LOAD_OFFSET" (PRELOA ;
2545:  R[87]=0    ;
2546:  !R[100] "GRIPPER_ID" 3 values ;
2547:  !If =100, ID Grippers Installed ;
2548:  !If =200, OD Grippers Installed ;
2549:  !If =300, OD 45 Degree Grippers ;
2550:  R[100]=100    ;
2551:  !--------------------------- ;
2552:   ;
2553:  !If using previous setup data ;
2554:  IF (R[71]=4857) THEN ;
2555:   ;
2556:  !--------------------------- ;
2557:  !1st: Height of Raw piece ;
2558:  R[190]=114.3    ;
2559:  !2nd: Height of Finish piece ;
2560:  R[191]=114.3    ;
2561:  !3rd: Infeed Height Offset ;
2562:  R[192]=(-300)    ;
2563:  !4th: Outfeed Height Offset ;
2564:  R[193]=(-40)    ;
2565:  !--------------------------- ;
2566:   ;
2567:  CALL CREATE_REG(R[190],R[191],R[192],R[193]) ;
2568:   ;
2569:  ENDIF ;
2570:   ;
2571:  !If new loading or offloading pos ;
2572:  !SET R[104] "IMPORT_LOADPOS" ;
2573:  !SET R[104]=1000, Otherwise NO ;
2574:  R[104]=1000    ;
2575:  IF (R[104]=1000) THEN ;
2576:  !R[260]=43, Preload Pos1 ;
2577:  !R[270]=44, Preload PosFinal ;
2578:  !R[300]=53, Offload PosFinal ;
2579:  !PR[43] Pre-Loading Pos1 ;
2580:  CALL CREATE_PR(43,167.537,(-62.622),133.47,103.2,89.276,102.077) ;
2581:  !PR[44] Final Loading Position ;
2582:  CALL CREATE_PR(44,167.72,(-63.542),190.442,103.416,89.263,102.281) ;
2583:  !PR[53] pre-Unloading Position ;
2584:  CALL CREATE_PR(53,(-129.189),92.632,169.217,170.145,(-88.272),(-171.356)) ;
2585:  !PR[54] Final Unloading Position ;
2586:  CALL CREATE_PR(54,(-126.007),92.8665,62.07,170.397,(-88.274),(-171.597)) ;
2587:  !PR[56] assitant Unloading preses ;
2588:  CALL CREATE_PR(56,(-133.84),95.467,273.686,(-177.134),(-88.249),175.184) ;
2589:  !PR[57] assitant Unloading preses ;
2590:  CALL CREATE_PR(57,(-135.964),108.085,344.284,(-177.144),(-88.245),175.194) ;
2591:  !PR[58] assitant Unloading preses ;
2592:  CALL CREATE_PR(58,296.854,360.959,378.47,(-91.75),(-.28),88.063) ;
2593:  ENDIF ;
2594:   ;
2595:  !---------------------------- ;
2596:  !SR[1] = "JOB_VAR_ID_GRIP" ;
2597:  !JOB_VAR_COMMON(R[103])'s value ;
2598:  !---------------------------- ;
2599:  !2By3 SR[1] INF, Max 18(Straight) ;
2600:  !R[103]=100 ;
2601:  !2By3 INF 45 Degree Diagonal Shif ;
2602:  !R[103]=110 ;
2603:  !---------------------------- ;
2604:  !3By4 SR[1] INF, Max 36(Straight) ;
2605:  !R[103]=150 ;
2606:  !3By4 INF 45 Degree Diagonal Shif ;
2607:  !R[103]=160 ;
2608:  !---------------------------- ;
2609:  !R[103] "JOB_PROFILE" Selection ;
2610:  R[103]=100    ;
2611:  CALL JOB_VAR_COMMON(R[103]) ;
2612:   ;
2613:  ENDIF ;
2614:   ;
2615:  JMP LBL[9999] ;
2616:   ;
2617:  !Job 100006970 Logic Ends ;
2618:  !--------------------------- ;
2619:   ;
2620:  LBL[7064] ;
2621:  !--------------------------- ;
2622:  !Shear Ring ;
2623:  !Item 101487064 , Rev A ;
2624:  !Last Modified: 2025-09-12 ;
2625:  !Modified by: Aaron ;
2626:  !1.00 IN Height ;
2627:  !2.73 IN ID, 3.215 IN OD ;
2628:  !ID Jaw # 1016 ;
2629:  !--------------------------- ;
2630:  IF (R[70]=7064) THEN ;
2631:   ;
2632:  !Define Parameters for INF/OTF ;
2633:  !R[105]=AR[1]=100, 2By3 Sheet ;
2634:  !R[105]=AR[1]=200, 3By4 Sheet ;
2635:  CALL JOB_VAR_SETUP(200) ;
2636:   ;
2637:  !--------------------------- ;
2638:  !Define Parameters for Job ;
2639:  !R[85] "INF_JAW_OFFSET"(Hgt) ;
2640:  R[85]=106.5    ;
2641:  !R[86] "INF_PICK_OFFSET" 50mm/sec ;
2642:  R[86]=60    ;
2643:  !R[87] "MAIN_LOAD_OFFSET" (PRELOA ;
2644:  R[87]=0    ;
2645:  !R[100] "GRIPPER_ID" 3 values ;
2646:  !If =100, ID Grippers Installed ;
2647:  !If =200, OD Grippers Installed ;
2648:  !If =300, OD 45 Degree Grippers ;
2649:  R[100]=100    ;
2650:  !--------------------------- ;
2651:   ;
2652:  !If using previous setup data ;
2653:  IF (R[71]=7064) THEN ;
2654:   ;
2655:  !--------------------------- ;
2656:  !1st: Height of Raw piece ;
2657:  R[190]=31.37    ;
2658:  !2nd: Height of Finish piece ;
2659:  R[191]=25.27    ;
2660:  !3rd: Infeed Height Offset ;
2661:  R[192]=(-50)    ;
2662:  !4th: Outfeed Height Offset ;
2663:  R[193]=(-93)    ;
2664:  !--------------------------- ;
2665:   ;
2666:  CALL CREATE_REG(R[190],R[191],R[192],R[193]) ;
2667:   ;
2668:  ENDIF ;
2669:   ;
2670:  !If new loading or offloading pos ;
2671:  !SET R[104] "IMPORT_LOADPOS" ;
2672:  !SET R[104]=1000, Otherwise NO ;
2673:  R[104]=1000    ;
2674:  IF (R[104]=1000) THEN ;
2675:  !R[260]=43, Preload Pos1 ;
2676:  !R[270]=44, Preload PosFinal ;
2677:  !R[300]=53, Offload PosFinal ;
2678:  !PR[43] Pre-Loading Pos1 ;
2679:  CALL CREATE_PR(43,168.572,(-60.923),352.023,67.102,89.464,65.289) ;
2680:  !PR[44] Final Loading Position ;
2681:  CALL CREATE_PR(44,168.293,(-61.788),363.901,79.248,89.446,77.416) ;
2682:  !PR[53] pre-Unloading Position ;
2683:  CALL CREATE_PR(53,(-125.093),95.886,36.656,173.09,(-88.208),(-174.916)) ;
2684:  !PR[54] Final Unloading Position ;
2685:  CALL CREATE_PR(54,(-124.357),95.73,13.108,173.17,(-88.209),(-174.985)) ;
2686:  !PR[56] assitant Unloading preses ;
2687:  CALL CREATE_PR(56,(-133.84),95.467,273.686,(-177.134),(-88.249),175.184) ;
2688:  !PR[57] assitant Unloading preses ;
2689:  CALL CREATE_PR(57,(-135.964),108.085,344.284,(-177.144),(-88.245),175.194) ;
2690:  !PR[58] assitant Unloading preses ;
2691:  CALL CREATE_PR(58,296.854,360.959,378.47,(-91.75),(-.28),88.063) ;
2692:  ENDIF ;
2693:   ;
2694:  !---------------------------- ;
2695:  !SR[1] = "JOB_VAR_ID_GRIP" ;
2696:  !JOB_VAR_COMMON(R[103])'s value ;
2697:  !---------------------------- ;
2698:  !2By3 SR[1] INF, Max 18(Straight) ;
2699:  !R[103]=100 ;
2700:  !2By3 INF 45 Degree Diagonal Shif ;
2701:  !R[103]=110 ;
2702:  !---------------------------- ;
2703:  !3By4 SR[1] INF, Max 36(Straight) ;
2704:  !R[103]=150 ;
2705:  !3By4 INF 45 Degree Diagonal Shif ;
2706:  !R[103]=160 ;
2707:  !---------------------------- ;
2708:  !R[103] "JOB_PROFILE" Selection ;
2709:  R[103]=150    ;
2710:  CALL JOB_VAR_COMMON(R[103]) ;
2711:   ;
2712:  ENDIF ;
2713:   ;
2714:  JMP LBL[9999] ;
2715:   ;
2716:  !Job 101487064 Logic Ends ;
2717:  !--------------------------- ;
2718:   ;
2719:  LBL[7132] ;
2720:  !--------------------------- ;
2721:  !Sleeve,Compression ;
2722:  !Item 101367132 , Rev A ;
2723:  !Last Modified: 2026-03-30 ;
2724:  !Modified by: Aaron ;
2725:  !2.99 IN Height ;
2726:  !2.88 IN ID, 3.9 IN OD, 6.5 Lbs W ;
2727:  !ID Jaw # 1016 ;
2728:  !--------------------------- ;
2729:  IF (R[70]=7132) THEN ;
2730:   ;
2731:  !Define Parameters for INF/OTF ;
2732:  !R[105]=AR[1]=100, 2By3 Sheet ;
2733:  !R[105]=AR[1]=200, 3By4 Sheet ;
2734:  CALL JOB_VAR_SETUP(100) ;
2735:   ;
2736:  !--------------------------- ;
2737:  !Define Parameters for Job ;
2738:  R[1]=1    ;
2739:  R[2]=0    ;
2740:  R[4]=0    ;
2741:  R[67]=40    ;
2742:  !R[85] "INF_JAW_OFFSET"(Hgt) ;
2743:  R[85]=111.4    ;
2744:  !R[86] "INF_PICK_OFFSET" 50mm/sec ;
2745:  R[86]=0    ;
2746:  !R[87] "MAIN_LOAD_OFFSET" (PRELOA ;
2747:  R[87]=0    ;
2748:  !R[100] "GRIPPER_ID" 3 values ;
2749:  !If =100, ID Grippers Installed ;
2750:  !If =200, OD Grippers Installed ;
2751:  !If =300, OD 45 Degree Grippers ;
2752:  R[100]=100    ;
2753:  !--------------------------- ;
2754:   ;
2755:  !If using previous setup data ;
2756:  IF (R[71]=7132) THEN ;
2757:   ;
2758:  !--------------------------- ;
2759:  !1st: Height of Raw piece ;
2760:  R[190]=84.2    ;
2761:  !2nd: Height of Finish piece ;
2762:  R[191]=75.95    ;
2763:  !3rd: Infeed Height Offset ;
2764:  R[192]=(-300)    ;
2765:  !4th: Outfeed Height Offset ;
2766:  R[193]=(-239)    ;
2767:  !--------------------------- ;
2768:   ;
2769:  CALL CREATE_REG(R[190],R[191],R[192],R[193]) ;
2770:   ;
2771:  ENDIF ;
2772:   ;
2773:  !If new loading or offloading pos ;
2774:  !SET R[104] "IMPORT_LOADPOS" ;
2775:  !SET R[104]=1000, Otherwise NO ;
2776:  R[104]=1000    ;
2777:  IF (R[104]=1000) THEN ;
2778:  !R[260]=43, Preload Pos1 ;
2779:  !R[270]=44, Preload PosFinal ;
2780:  !R[300]=53, Offload PosFinal ;
2781:  !PR[43] Pre-Loading Pos1 ;
2782:  CALL CREATE_PR(43,167.348,(-60.809),341.996,144.299,89.137,142.832) ;
2783:  !PR[44] Final Loading Position ;
2784:  CALL CREATE_PR(44,167.772,(-61.005),377.015,144.427,89.137,142.97) ;
2785:  !PR[53] pre-Unloading Position ;
2786:  CALL CREATE_PR(53,(-126.517),93.375,44.616,169.258,(-88.267),(-170.592)) ;
2787:  !PR[54] Final Unloading Position ;
2788:  CALL CREATE_PR(54,(-125.31),93.435,4.826,169.28,(-88.267),(-170.606)) ;
2789:  !PR[56] assitant Unloading preses ;
2790:  CALL CREATE_PR(56,(-133.84),95.467,273.686,(-177.134),(-88.249),175.184) ;
2791:  !PR[57] assitant Unloading preses ;
2792:  CALL CREATE_PR(57,(-135.964),108.085,344.284,(-177.144),(-88.245),175.194) ;
2793:  !PR[58] assitant Unloading preses ;
2794:  CALL CREATE_PR(58,296.854,360.959,378.47,(-91.75),(-.28),88.063) ;
2795:  ENDIF ;
2796:   ;
2797:  !---------------------------- ;
2798:  !SR[1] = "JOB_VAR_ID_GRIP" ;
2799:  !JOB_VAR_COMMON(R[103])'s value ;
2800:  !---------------------------- ;
2801:  !2By3 SR[1] INF, Max 18(Straight) ;
2802:  !R[103]=100 ;
2803:  !2By3 INF 45 Degree Diagonal Shif ;
2804:  !R[103]=110 ;
2805:  !---------------------------- ;
2806:  !3By4 SR[1] INF, Max 36(Straight) ;
2807:  !R[103]=150 ;
2808:  !3By4 INF 45 Degree Diagonal Shif ;
2809:  !R[103]=160 ;
2810:  !---------------------------- ;
2811:  !R[103] "JOB_PROFILE" Selection ;
2812:  R[103]=100    ;
2813:  CALL JOB_VAR_COMMON(R[103]) ;
2814:   ;
2815:  ENDIF ;
2816:   ;
2817:  JMP LBL[9999] ;
2818:   ;
2819:  !Job 101367132 Logic Ends ;
2820:  !--------------------------- ;
2821:   ;
2822:  LBL[7920] ;
2823:  !--------------------------- ;
2824:  !Wedge ;
2825:  !Item 102745613 , Rev A ;
2826:  !Last Modified: 2026-01-25 ;
2827:  !Modified by: Aaron ;
2828:  !2.40 IN Height ;
2829:  !2.01 IN ID, 3.46 IN OD ;
2830:  !ID Jaw # 1031 ;
2831:  !--------------------------- ;
2832:  IF (R[70]=7920) THEN ;
2833:   ;
2834:  !Define Parameters for INF/OTF ;
2835:  !R[105]=AR[1]=100, 2By3 Sheet ;
2836:  !R[105]=AR[1]=200, 3By4 Sheet ;
2837:  CALL JOB_VAR_SETUP(200) ;
2838:   ;
2839:  !--------------------------- ;
2840:  !Define Parameters for Job ;
2841:  !R[85] "INF_JAW_OFFSET"(Hgt) ;
2842:  R[85]=10    ;
2843:  !R[86] "INF_PICK_OFFSET" 50mm/sec ;
2844:  R[86]=5    ;
2845:  !R[87] "MAIN_LOAD_OFFSET" (PRELOA ;
2846:  R[87]=0    ;
2847:  !R[100] "GRIPPER_ID" 3 values ;
2848:  !If =100, ID Grippers Installed ;
2849:  !If =200, OD Grippers Installed ;
2850:  !If =300, OD 45 Degree Grippers ;
2851:  R[100]=100    ;
2852:  !--------------------------- ;
2853:   ;
2854:  !If using previous setup data ;
2855:  IF (R[71]=7920) THEN ;
2856:   ;
2857:  !--------------------------- ;
2858:  !1st: Height of Raw piece ;
2859:  R[190]=63.5    ;
2860:  !2nd: Height of Finish piece ;
2861:  R[191]=60.96    ;
2862:  !3rd: Infeed Height Offset ;
2863:  R[192]=(-13)    ;
2864:  !4th: Outfeed Height Offset ;
2865:  !Changing 1st Level Offset to ;
2866:  R[193]=(-26)    ;
2867:   ;
2868:  !Changing 2nd Level Offset to ;
2869:  R[194]=(-26)    ;
2870:   ;
2871:  !Changing 3rd Level Offset to ;
2872:  R[195]=(-26)    ;
2873:   ;
2874:  CALL GN_OUTFEED_COMPENSATE(R[193],R[194],R[195]) ;
2875:  !--------------------------- ;
2876:   ;
2877:  CALL CREATE_REG(R[190],R[191],R[192],R[193]) ;
2878:   ;
2879:  ENDIF ;
2880:   ;
2881:  !If new loading or offloading pos ;
2882:  !SET R[104] "IMPORT_LOADPOS" ;
2883:  !SET R[104]=1000, Otherwise NO ;
2884:  R[104]=1000    ;
2885:  IF (R[104]=1000) THEN ;
2886:  !R[260]=43, Preload Pos1 ;
2887:  !R[270]=44, Preload PosFinal ;
2888:  !R[300]=53, Offload PosFinal ;
2889:  !PR[43] Pre-Loading Pos1 ;
2890:  CALL CREATE_PR(43,168.34,(-59.237),294.359,129.783,89.102,128.057) ;
2891:  !PR[44] Final Loading Position ;
2892:  CALL CREATE_PR(44,168.503,(-59.508),309.049,129.895,89.101,128.164) ;
2893:  !PR[53] pre-Unloading Position ;
2894:  CALL CREATE_PR(53,(-127.892),94.224,101.759,162.89,(-88.35),(-164.668)) ;
2895:  !PR[54] Final Unloading Position ;
2896:  CALL CREATE_PR(54,(-126.656),94.628,56.811,162.912,(-88.351),(-164.695)) ;
2897:  !PR[56] assitant Unloading preses ;
2898:  CALL CREATE_PR(56,(-133.84),95.467,273.686,(-177.134),(-88.249),175.184) ;
2899:  !PR[57] assitant Unloading preses ;
2900:  CALL CREATE_PR(57,(-135.964),108.085,344.284,(-177.144),(-88.245),175.194) ;
2901:  !PR[58] assitant Unloading preses ;
2902:  CALL CREATE_PR(58,296.854,360.959,378.47,(-91.75),(-.28),88.063) ;
2903:  ENDIF ;
2904:   ;
2905:  !---------------------------- ;
2906:  !SR[1] = "JOB_VAR_ID_GRIP" ;
2907:  !JOB_VAR_COMMON(R[103])'s value ;
2908:  !---------------------------- ;
2909:  !2By3 SR[1] INF, Max 18(Straight) ;
2910:  !R[103]=100 ;
2911:  !2By3 INF 45 Degree Diagonal Shif ;
2912:  !R[103]=110 ;
2913:  !---------------------------- ;
2914:  !3By4 SR[1] INF, Max 36(Straight) ;
2915:  !R[103]=150 ;
2916:  !3By4 INF 45 Degree Diagonal Shif ;
2917:  !R[103]=160 ;
2918:  !---------------------------- ;
2919:  !R[103] "JOB_PROFILE" Selection ;
2920:  R[103]=150    ;
2921:  CALL JOB_VAR_COMMON(R[103]) ;
2922:   ;
2923:  ENDIF ;
2924:   ;
2925:  JMP LBL[9999] ;
2926:   ;
2927:  !Job 101477920 Logic Ends ;
2928:  !--------------------------- ;
2929:   ;
2930:  LBL[7937] ;
2931:  !--------------------------- ;
